(* CODESYS project OC_Core.library
   DefaultNamespace: OC_Core
   DocFormat: reStructuredText
   Description: Open Commissioning TwinCAT Core Library
   Author: SpiraTec AG
   Title: OC_Core
   Version: 1.1.0
   Company: Open Commissioning
   Placeholder: OC_Core

Project tree, tasks and I/O mapping:
  libraries: Tc2_Math, * (Beckhoff Automation GmbH); Tc2_Standard, * (Beckhoff Automation GmbH); Tc2_System, * (Beckhoff Automation GmbH); Tc2_Utilities, * (Beckhoff Automation GmbH); Tc3_Module, * (Beckhoff Automation GmbH); TcUnit, * (www.tcunit.org)
  Common/
    AdsMessageHandler/
      function block FB_AdsMessageHandler [ST]: bIsAdsMessageReadValid, bIsAdsMessageWriteValid, CreateAdsReadMessage, CreateAdsWriteMessage, LogAdsMessage, SendReadResponse, SendWriteResponse, stAdsMessageRead, stAdsMessageWrite
      data type ST_AdsMessage
    Components/
      function block FB_Clock [ST]
      function block FB_ClockAdvanced [ST]
      function block FB_DriveControl [ST]: bIsMoving, bIsPositionReached, fAccMax, fPosition, fPositionLimitMax, fPositionLimitMin, fTolerance, fVelocity, MoveAbsolute, MoveVelocity, Stop
      function block FB_Heater [ST]: FB_init, fValue, InitRun
      function block FB_MoveAbsolute [ST]: bIsReached, fPosition, fVelocity
      function block FB_MoveVelocity [ST]: bIsReached, fAcc, fVelocity
      function block FB_Ping [ST]: InitRun
    FileIo/
      data type E_FileIoState
      function block FB_FileIO [ST]: nBytesRead, nErrorId, Read, sNetId, sPath, Write
    Links/
      function block FB_LinkDataByte [ST]: GetLinkControlData, SetLinkStatusData
      function block FB_LinkDataDWord [ST]: GetLinkControlData, SetLinkStatusData
      function block FB_LinkDataLWord [ST]: GetLinkControlData, SetLinkStatusData
      function block FB_LinkDataReal [ST]: GetLinkControlData, SetLinkStatusData
      function block FB_LinkDataWord [ST]: GetLinkControlData, SetLinkStatusData
      function block FB_LinkDevice [ST]: GetControl, SetStatus
    RecordData/
      function block FB_RecordData [ST]: CmpIGrp, CmpInvokeId, CmpIOffs, DataValid, FB_init, GetReadIndication, GetWriteIndication, SendReadResponse, SendWriteResponse, Subscribe
      interface I_RecordData: GetReadIndication, GetWriteIndication, SendReadResponse, SendWriteResponse, Subscribe
      data type ST_RecordIdent
    System/
      data type E_ControllerType
      function F_IsSystemValid [ST]
      function F_LogError [ST]
      function F_LogMessage [ST]
      function F_LogWarning [ST]
      function block FB_Base [ST]
      function block FB_System [ST]: bDebug, bVerbose, eControllerType, fDeltaTime, fTimeScaling, InitRun
      global variables GVL_Core
    Utils/
      data type E_NetworkByteOrder
      function F_Clamp01 [ST]
      function F_Compare [ST]
      function F_GetHByte [ST]
      function F_GetLByte [ST]
      function F_InverBytesOrder [ST]
      function F_Norm [ST]
      function F_ScaleLREAL [ST]
      function F_Sign [ST]
      data type ST_ScaleConfig
  Devices/
    Basic/
      function block FB_Button [ST]
      function block FB_Cylinder [ST]
      function block FB_Device [ST]
      function block FB_DeviceByte [ST]
      function block FB_DeviceDWord [ST]
      function block FB_DeviceLWord [ST]
      function block FB_DeviceReal [ST]
      function block FB_DeviceWord [ST]
      function block FB_Drive [ST]
      function block FB_Lamp [ST]
      function block FB_Lock [ST]
      function block FB_Panel [ST]
      function block FB_Reader [ST]
      function block FB_Robot [ST]: ConnectJoints, GetJointsTarget, SetJointsStatus
      function block FB_SensorAnalog [ST]
      function block FB_SensorBinary [ST]
      function block FB_Switch [ST]
    Drives/
      Encoder/
        function block FB_Encoder [ST]: ControlLogic, InitRun
        data type ST_EncoderConfig
      FB_DS402/
        data type E_ControlMode
        data type E_DS402State
        function block FB_DS402 [ST]: AssignAddress, ControlLogic, eState, GetControlData, InitRun, PositionMode, SetStatusData, SpeedMode
        function block FB_DS402FSM [ST]: eState, IsDisableOperation, IsDisableVoltage, IsEnableOperation, IsFaultReset, IsQuickStop, IsShutdown, IsSwitchOn, nControl, nStatus, S0_NotReadyToSwitchOn, S1_SwitchOnDisabled, S2_ReadyToSwitchOn, S3_SwitchedOn, S4_OperationEnabled, S5_Fault, S6_FaultReactionActive, S7_QuickStopActive
        data type ST_DS402_6040h_ControlWord
        data type ST_DS402_6041h_StatusWord
        data type ST_DS402Config
      FB_SimMovidrive/
        data type E_SimMovidriveMode
        function block FB_SimMovidrivePDO12 [ST]: AssignProcessData, ControlLogic, GetControlData, GetControlMode, InitRun, SetStatusData
        data type ST_SimMovidriveConfig
        data type ST_SimMovidriveControlData
        data type ST_SimMovidriveStatusData
      FB_SimMovitrac/
        data type E_SimMovitracAssign
        function block FB_SimMovitrac [ST]: AssignProcessData, ControlLogic, GetControlData, InitRun, SetStatusData
        function block FB_SimMovitracB [ST]: AssignProcessData, ControlLogic, GetControlData, InitRun, SetStatusData
        function block FB_SimMovitracLTEB [ST]: ControlLogic, InitRun
        data type ST_SimMovitracConfig
        data type ST_SimMovitracControlData
        data type ST_SimMovitracStatusData
      FB_SimMovitracFSM/
        data type E_SimMovitracState
        function block FB_SimMovitracFSM [ST]: ControllerInhibit, Enable, Halt, HoldControl, nState, RapidStop
      FB_Starter/
        function block FB_Starter [ST]: AssignProcessData, ControlLogic, GetControlData, InitRun, SetStatusData
        data type ST_StarterConfig
        data type ST_StarterControlData
        data type ST_StarterStatusData
    Safety/
      function block FB_EuchnerMGB [ST]
      function block FB_EuchnerSTP [ST]
  Test/
    Common/
      function block FB_AdsMessageHandler_Test [ST]: TestCaseRead, TestCaseWrite
      function block FB_Clamp01_Test [ST]: TestCase
      function block FB_Compare_Test [ST]: TestCase
      function block FB_GetByte_Test [ST]: TestGetHByte, TestGetLByte
      function block FB_InverBytesOrder_Test [ST]: TestDWord, TestLWord, TestWord
      function block FB_Norm_Test [ST]: TestCase
      function block FB_RecordData_Test [ST]: TestAutoResponseReadMessage, TestAutoResponseWriteMessage, TestCaseCompare, TestCasesCompare, TestGetReadIndication, TestGetWriteIndication, TestSendReadResponse, TestSendWriteResponse
      function block FB_Scale_Test [ST]: TestCase, TestInputValidation
      function block FB_Sign_Test [ST]: TestCase
      function block FB_System_Test [ST]: TestInitialization, TestProperties
    Components/
      function block FB_DriveControl_Test [ST]: TestCaseMoveAbsolute, TestCaseMoveVelocity, TestCaseMoveVelocityLimits, TestProperties, TestStop
      function block FB_Heater_Test [ST]: TestLimits, TestState, TestValueChange
      function block FB_MoveAbsolute_Test [ST]: TestCaseMoveTo
      function block FB_MoveVelocity_Test [ST]: TestCaseMove
    Devices/
      function block FB_Button_Test [ST]
      function block FB_Cylinder_Test [ST]
      function block FB_Device_Test [ST]
      function block FB_DeviceByte_Test [ST]
      function block FB_DeviceDWord_Test [ST]
      function block FB_DeviceLWord_Test [ST]
      function block FB_DeviceReal_Test [ST]
      function block FB_DeviceWord_Test [ST]
      function block FB_Drive_Test [ST]
      function block FB_Lamp_Test [ST]
      function block FB_Lock_Test [ST]
      function block FB_Panel_Test [ST]
      function block FB_Reader_Test [ST]
      function block FB_Robot_Test [ST]: TestGetJoint, TestSetJoint
      function block FB_SensorAnalog_Test [ST]
      function block FB_SensorBinary_Test [ST]
      function block FB_Switch_Test [ST]
    Drives/
      function block FB_DS402_Test [ST]: EnableSequence, TestEnable, TestEnableSTO, TestPositionMode, TestSpeedDriveFactor, TestSpeedMode, TestSpeedModeEncoder, TestSpeedModeLinkOutput, TestSpeedModeModulo, TestSpeedModeOffset
      function block FB_DS402FSM_Test [ST]: GetDisableCommand, GetDisableVoltageCommand, GetEnableCommand, GetQuickStopCommand, GetShotdownCommand, GetSwitchOnCommand, TestEnableSequence, TestState_S0, TestState_S1, TestState_S2, TestState_S3, TestState_S4, TestState_S5, TestState_S6, TestState_S7
      function block FB_Encoder_Test [ST]: TestCase_Encoder
      function block FB_SimMovidriveFSM_Test [ST]: TestState
      function block FB_SimMovidrivePDO12_Test [ST]: Test_AssignProcessData, Test_GetControlData, Test_GetControlDataSWAP, Test_GetControlMode, Test_SetStatusData, Test_SetStatusDataSWAP
      function block FB_SimMovitrac_Test [ST]: Test_Movitrac
      function block FB_SimMovitracB_Test [ST]: TestCase_SimMovitracB
      function block FB_SimMovitracLTEB_Test [ST]: Test_DriveNotReady, Test_DriveReady, Test_DriveRunningBwd, Test_DriveRunningFwd
      function block FB_Starter_Test [ST]: Test_AssignProcessData, Test_DriveNoMovement, Test_DriveRunningCcw, Test_DriveRunningCw, Test_GetControlData, Test_GetControlDataSWAP, Test_SetStatusData, Test_SetStatusDataSWAP
    Safety/
      function block FB_Euchner_MGB_Test [ST]: Test_Button1, Test_Button2, Test_Button3, Test_Button4, Test_DoorClosed_Locked, Test_DoorClosed_NoLock, Test_DoorOpen, Test_Lamp1, Test_Lamp2, Test_Lamp3, Test_Lamp4
      function block FB_Euchner_STP_Test [ST]: Test_DoorClosedAndLocked, Test_DoorClosedAndUnlocked, Test_DoorOpen, Test_LampGN, Test_LampRD
    program PRG_TEST [ST]
*)

// Common/AdsMessageHandler/ST_AdsMessage
TYPE ST_AdsMessage :
STRUCT
	tNetID			: T_AmsNetID;
	tPort			: T_AmsPort;
	nInvokeID		: UDINT;
	nIdxGrp			: UDINT;
	nIdxOffs		: UDINT;
	nLength			: UDINT;
	nResult			: UDINT;
	aData			: ARRAY[0..239] OF BYTE;
END_STRUCT
END_TYPE

// Common/FileIo/E_FileIoState
{attribute 'conditionalshow'}
TYPE E_FileIoState :
(
	READY := 0,
	OPEN,
	CREATE,
	READ,
	WRITE,
	CLOSE,
	ERROR
);
END_TYPE

// Common/RecordData/ST_RecordIdent
TYPE ST_RecordIdent :
STRUCT
	nPort  			: T_AmsPort; //ADS-Port of the Profinet Device. Ignored when using PLCSIM Advanced
	nSlot			: UINT; //Slotnumber of the Profinet Device. Ignored when using PLCSIM Advanced
	nSubSlot		: UINT; //Subslotnumber of the Profinet Device. Ignored when using PLCSIM Advanced
	nPlcId			: UINT; //Identifier of the PLC when using PLCSIM Advanced
	nHardwareId		: UINT; //Hardware-ID of the device when using PLCSIM Advanced
END_STRUCT
END_TYPE

// Common/System/E_ControllerType
{attribute 'qualified_only'}
{attribute 'strict'}
TYPE E_ControllerType :
(
	NotDefined := 0,
	PlcSimAdvanced := 1
);
END_TYPE

// Common/Utils/E_NetworkByteOrder
{attribute 'qualified_only'}
{attribute 'strict'}
TYPE E_NetworkByteOrder :
(
	BigEndian := 0, //Big Endian (MOTOROLA)
	LittleEndian := 1 //Little Endian (Intel)	
);
END_TYPE

// Common/Utils/ST_ScaleConfig
{attribute 'pack_mode' := '0'} 
TYPE ST_ScaleConfig :
STRUCT
	fInputMin 	: LREAL := 0;
	fInputMax 	: LREAL := 100;
	fOutputMin 	: LREAL := 0;
	fOutputMax 	: LREAL := 65535;
END_STRUCT
END_TYPE

// Devices/Drives/Encoder/ST_EncoderConfig
TYPE ST_EncoderConfig :
STRUCT
	bIsIntegral   			: BOOL := FALSE;  //Integrate input value
	fNumerator 	  			: REAL := 0.0001; //[unit/INC]
	fDenominator  			: REAL := 1.0; 	// Scaling
	fModulo 	  			: REAL := 0; 	 	// Base divisor for modulo calculation [unit]; If not used set to 0.0	
	fInputFactor  			: REAL := 1.0; 
	fOutputFactor 			: REAL := 1.0;
	bInvertIncrementValue 	: BOOL;
END_STRUCT
END_TYPE

// Devices/Drives/FB_DS402/E_ControlMode
{attribute 'qualified_only'}
{attribute 'strict'}
TYPE E_ControlMode :
(
	Position 	:= 0,
	Speed	 	:= 1
)
BYTE;
END_TYPE

// Devices/Drives/FB_DS402/E_DS402State
{attribute 'qualified_only'}
{attribute 'strict'}
{attribute 'conditionalshow'}
TYPE E_DS402State :
(
	S0_NotReadyToSwitchOn,
	S1_SwitchOnDisabled,
	S2_ReadyToSwitchOn,
	S3_SwitchedOn,
	S4_OperationEnabled,
	S5_Fault,
	S6_FaultReactionActive,
	S7_QuickStopActive
);
END_TYPE

// Devices/Drives/FB_DS402/ST_DS402_6040h_ControlWord
{attribute 'pack_mode' := '1'}
TYPE ST_DS402_6040h_ControlWord :
STRUCT
	b0_SwitchOn 					: BIT;
	b1_EnableVoltage				: BIT;
	b2_QuickStop					: BIT;
	b3_EnableOperation				: BIT;
	b4_OperationModeSpecific		: BIT;
	b5_OperationModeSpecific		: BIT;
	b6_OperationModeSpecific		: BIT;
	b7_FaultReset					: BIT;
	b8_Reserved						: BIT;
	b9_Reserved						: BIT;
	b10_Reserved					: BIT;
	b11_Reserved					: BIT;
	b12_Reserved					: BIT;
	b13_Reserved					: BIT;
	b14_Reserved					: BIT;
	b15_Reserved					: BIT;
END_STRUCT
END_TYPE

// Devices/Drives/FB_DS402/ST_DS402_6041h_StatusWord
{attribute 'pack_mode' := '1'}
TYPE ST_DS402_6041h_StatusWord :
STRUCT
	b0_ReadyToSwitchOn 				: BIT; 
	b1_SwitchedOn 					: BIT; 
	b2_OperationEnabled 			: BIT; 
	b3_Fault						: BIT; 
	b4_VoltageEnabled				: BIT; 
	b5_QuickStop					: BIT;
	b6_SwitchOnDisabled				: BIT; 
	b7_Warning						: BIT; 
	b8_Synchranisation				: BIT; 
	b9_Remote						: BIT;
	b10_TargetReached				: BIT;
	b11_InternalLimitActive			: BIT; 
	b12_OperationModeSpecific		: BIT; 
	b13_OperationModeSpecific		: BIT; 
	b14_OperationModeSpecific		: BIT; 
	b15_ClosedLoopActive			: BIT;	
END_STRUCT
END_TYPE

// Devices/Drives/FB_DS402/ST_DS402Config
TYPE ST_DS402Config :
STRUCT	
	eControlMode 			: E_ControlMode := E_ControlMode.Position;
	eLinkControlMode 		: E_ControlMode := E_ControlMode.Position;
	fReferenceVelocity 		: REAL := 1000.0;
	fPositionOffset			: REAL := 0.0;	
	
	fEncoderNumerator		: REAL := 0.0001; //[unit/INC]
	fEncoderDenominator		: REAL := 1.0; //Scaling
	fEncoderModulo			: REAL := 0; //[unit]	
	
	fGearFactor				: REAL := 1.0;
	fEncoderOutputFactor	: REAL := 1.0;
	fLinkOutputFactor 		: REAL := 1.0;
	
	bSwapProcessData		: BOOL; //SWAP Process Data from/to FIELDBUS
END_STRUCT
END_TYPE

// Devices/Drives/FB_SimMovidrive/E_SimMovidriveMode
{attribute 'qualified_only'}
{attribute 'strict'}
TYPE E_SimMovidriveMode :
(
	Idle 	:= 0,
	Jog	 	:= 1,
	Ref		:= 2,
	Auto	:= 3
)BYTE;
END_TYPE

// Devices/Drives/FB_SimMovidrive/ST_SimMovidriveConfig
{attribute 'pack_mode' := '0'}
TYPE ST_SimMovidriveConfig :
STRUCT
	nSoftwareLimitMin	: DINT := -2147483648;	//Position limit minimum in LU
	nSoftwareLimitMax	: DINT := 2147483647;	//Position limit maximum in LU
	fDecCoastStop		: REAL := 10000.0;		//Deceleration for coast/brake stop in LU/s^2
	fDecRapidStop		: REAL := 10000.0;		//Deceleration for emergency stop in LU/s^2
	fDecRampStop		: REAL := 1000.0;		//Decceleration limit (bus stop) in LU/s^2
	fRatioVelocity		: REAL := 1.0;			//Ratio for setpoint velocity
	fRatioAccDec		: REAL := 1.0;			//Ratio for setpoint acceleration/deceleration
	fRatioPosition		: REAL := 0.001;		//Ratio for position output
	nJerk				: INT := 0;				//Jerk from 0 to 100%
	bSwapProcessData	: BOOL;					//SWAP Process Data from/to FIELDBUS
END_STRUCT
END_TYPE

// Devices/Drives/FB_SimMovidrive/ST_SimMovidriveControlData
{attribute 'pack_mode' := '1'}
TYPE ST_SimMovidriveControlData :
STRUCT
	bControllerInhibit		: BIT;	//0			0 = Enable, 1 = Inhibit controller, activate brake
	bRapidStop				: BIT;	//1			0 = Rapid stop, 1 = Enable
	bStop					: BIT;	//2			0 =  Stop at integrator ramp or process ramp, 1 = Enable
	bReserved3				: BIT;	//3			Currently not used
	bReserved4				: BIT;	//4			Currently not used
	bReserved5				: BIT;	//5			Currently not used
	bResetFAULT		  		: BIT;	//6			0 → 1 = Reset fault 
	bReserved7				: BIT;	//7			Currently not used	                            
	bStart					: BIT;	//8			1 = Enable Positioning / Referencing 
	bJog1					: BIT;	//9			1 = Enable Jog+
	bJog2					: BIT;	//10		1 = Enable Jog-
	bModeLow				: BIT;	//11		1 = Mode Jogging or Positioning (in combination with mode high)
	bModeHigh				: BIT;	//12		1 = Mode Referencing or Positioning (in combination with mode low)
	bReserved13				: BIT;	//13		Currently not used
	bReserved14				: BIT;	//14		Currently not used
	bReserved15				: BIT;	//15		Currently not used
	nTargetPosition			: DINT;	//16..47	Target position
	nVelocity				: UINT; //48..63	Velocity
	nAcceleration			: UINT; //64..79	Acceleration
	nDeceleration			: UINT; //80..95	Deceleration			
END_STRUCT
END_TYPE

// Devices/Drives/FB_SimMovidrive/ST_SimMovidriveStatusData
{attribute 'pack_mode' := '1'}
TYPE ST_SimMovidriveStatusData :
STRUCT
	bMotorTurning			: BIT;	//0			1 = Motor is turning
	bInverterReady			: BIT;	//1			1 = Inverter is ready
	bReferenced				: BIT;	//2			1 = Drive is referenced
	bTargetPositionReached	: BIT;	//3			1 = Target position reached
	bBrakeReleased			: BIT;	//4			1 = Brake is released
	bError					: BIT;	//5			1 = Error
	bLimitSwitchCW		  	: BIT;	//6			1 = Limit switch clock wise reached 
	bLimitSwitchCCW			: BIT;	//7			1 = Limit switch counter clock wise reached 	                            
	nStatus					: BYTE;	//8..15		Status / Errorcode
	nActPosition			: DINT; //16..47	Actual position
	nActVelocity			: UINT; //48..63	Actual velocity
	nActCurrent				: UINT; //64..79	Acutal current
	nActUnit				: UINT; //80..95	Actual unit utilization
END_STRUCT
END_TYPE

// Devices/Drives/FB_SimMovitrac/E_SimMovitracAssign
{attribute 'qualified_only'}
{attribute 'strict'}
TYPE E_SimMovitracAssign :
(
	ProcessData1 := 0,
	ProcessData2 := 2,
	ProcessData3 := 4,
	NoAssignment := 99
)DWORD;
END_TYPE

// Devices/Drives/FB_SimMovitrac/ST_SimMovitracConfig
TYPE ST_SimMovitracConfig :
STRUCT
	fDecCoastStop		: REAL := 200.0;	//Deceleration for coast/brake stop in ms. Reference speed is 3000 rpm.
	fDecRapidStop		: REAL := 500.0;	//Deceleration for emergency stop in ms. Reference speed is 3000 rpm.
	fProcessRamp		: REAL := 1000.0;	//Acc/Dec in ms when ramp via bus is not assigned. Reference speed is 3000 rpm.
	fGearFactor			: REAL := 1.0;		//Ratio for velocity output
	fReferenceVelocity	: REAL := 3000.0;

	nCtrlAssign			: E_SimMovitracAssign := E_SimMovitracAssign.ProcessData1; //Control word assignment
	nSpeedAssign		: E_SimMovitracAssign := E_SimMovitracAssign.ProcessData2; //Speed setpoint assignment
	nRampAssign			: E_SimMovitracAssign := E_SimMovitracAssign.NoAssignment; //Ramp setpoint assignment
	nStatusAssign		: E_SimMovitracAssign := E_SimMovitracAssign.ProcessData1; //Status word assignment
	nSpeedActAssign		: E_SimMovitracAssign := E_SimMovitracAssign.ProcessData2; //Actual speed assignment
	
	bSwapProcessData	: BOOL; //SWAP Process Data from/to FIELDBUS
END_STRUCT
END_TYPE

// Devices/Drives/FB_SimMovitrac/ST_SimMovitracControlData
{attribute 'pack_mode' := '1'}
TYPE ST_SimMovitracControlData :
STRUCT
	bControllerInhibit		: BIT;	//0			0 = Enable, 1 = Inhibit controller, activate brake
	bRapidStop				: BIT;	//1			0 = Rapid stop, 1 = Enable
	bStop					: BIT;	//2			0 =  Stop at integrator ramp or process ramp, 1 = Enable
	bReserved3				: BIT;	//3			Currently not used
	bReserved4				: BIT;	//4			Currently not used
	bReserved5				: BIT;	//5			Currently not used
	bResetFAULT		  		: BIT;	//6			0 → 1 = Reset fault 
	bReserved7				: BIT;	//7			Currently not used	                            
	bDirectionMotorPoti		: BIT;	//8			0 = CW, 1 = CCW 
	bMotorPotiUp			: BIT;	//9			1 = Increase poti value
	bMotorPotiDown			: BIT;	//10		1 = Decrease poti value
	bFixedInternalSetpoints	: BIT;	//11		1 = Fixed internal setpoints
	bFixedInternalSetp1		: BIT;	//12		1 = Fixed internal setpoint 1
	bFixedSetpSwitchover	: BIT;	//13		1 = Fixed setpoint switchover
	bReserved14				: BIT;	//14		Currently not used
	bReserved15				: BIT;	//15		Currently not used
	nSetpointSpeed			: INT; 	//			Setpoint speed in 0.2 rpm
	nRamp					: UINT; //			Ramp in ms			
END_STRUCT
END_TYPE

// Devices/Drives/FB_SimMovitrac/ST_SimMovitracStatusData
{attribute 'pack_mode' := '1'}
TYPE ST_SimMovitracStatusData :
STRUCT
	bEnableOutputStage		: BIT;	//0			1 = Output stage enabled
	bInverterReady			: BIT;	//1			1 = Inverter is ready
	bPoDataEnable			: BIT;	//2			1 = PO data enabled
	bReserved3				: BIT;	//3			Currently not used
	bReserved4				: BIT;	//4			Currently not used
	bError					: BIT;	//5			1 = Error
	bReserved6		  		: BIT;	//6			Currently not used
	bReserved7				: BIT;	//7			Currently not used
	nStatus					: BYTE;	//8..15		Status / Errorcode
	nActSpeed				: INT;	//			Actual speed in 0.2 rpm
END_STRUCT
END_TYPE

// Devices/Drives/FB_SimMovitracFSM/E_SimMovitracState
{attribute 'qualified_only'}
{attribute 'strict'}
{attribute 'conditionalshow'}
TYPE E_SimMovitracState :
(
	ControllerInhibit := 1,
	RapidStop := 2,
	Halt := 3,
	HoldControl := 4,
	Enable := 5
);
END_TYPE

// Devices/Drives/FB_Starter/ST_StarterConfig
{attribute 'pack_mode' := '1'}
TYPE ST_StarterConfig:
STRUCT
	fVelocity			: REAL := 100; 	// mm
	fAcceleration		: REAL := 500; 	// deg/s2
	fDeceleration		: REAL := 500; 	// deg/s2		
	bSwapProcessData	: BOOL; //SWAP Process Data from/to FIELDBUS
END_STRUCT
END_TYPE

// Devices/Drives/FB_Starter/ST_StarterControlData
{attribute 'pack_mode' := '1'}
TYPE ST_StarterControlData:
	STRUCT
		MotorCW           			: BIT; 		//0  
		MotorCCW	      			: BIT; 		//1  
		BrakeActuation				: BIT; 		//2  
		TripReset          			: BIT; 		//3  
		EmergStart        			: BIT; 		//4  
		SelfTest	      			: BIT; 		//5  
		Reserve06          			: BIT; 		//6  
		Reserve07		   			: BIT; 		//7 
		Reserve10		   			: BIT; 		//08  
		Reserve11		   			: BIT; 		//09  
		Reserve12		   			: BIT; 		//10  
		Reserve13		   			: BIT; 		//11  
		Reserve14		   			: BIT; 		//12  
		Reserve15		   			: BIT; 		//13  
		Reserve16		   			: BIT; 		//14  
		DisQuickStop	   			: BIT; 		//15   
	END_STRUCT
END_TYPE

// Devices/Drives/FB_Starter/ST_StarterStatusData
{attribute 'pack_mode' := '1'}
TYPE ST_StarterStatusData:
	STRUCT
		Ready           			: BIT; 		//0  
		MotorON		      			: BIT; 		//1  
		GroupFault					: BIT; 		//2  
		GroupWarn          			: BIT; 		//3  
		Input1	        			: BIT; 		//4  
		Input2		      			: BIT; 		//5  
		Input3          			: BIT; 		//6  
		Input4			   			: BIT; 		//7 
		MotorCurrent0	   			: BIT; 		//08  
		MotorCurrent1	   			: BIT; 		//09  
		MotorCurrent2	   			: BIT; 		//10  
		MotorCurrent3	   			: BIT; 		//11  
		MotorCurrent4	   			: BIT; 		//12  
		MotorCurrent5	   			: BIT; 		//13  
		ManualLocalMode	   			: BIT; 		//14  
		RampOperation	   			: BIT; 		//15  
	END_STRUCT
END_TYPE

// Common/System/GVL_Core
{attribute 'qualified_only'}
{attribute 'conditionalshow'}
VAR_GLOBAL	
	refSystem 			: REFERENCE TO FB_System;		
END_VAR

// Common/AdsMessageHandler/FB_AdsMessageHandler
(*ADS Message Handler is responsible for indication of the ADS Read/Write messages for local NetId and generation of the response message*)
FUNCTION_BLOCK FB_AdsMessageHandler
VAR_INPUT
	bDisable 				: BOOL;	//Deactivate cyclical execution
	bLog					: BOOL;	//Log ADS messages data in the console
	bVerbose				: BOOL; //Log Verbose information in the console
END_VAR

VAR	
	fbAdsWriteIndicator 	: AdsWriteInd;	
	fbAdsReadIndicator 		: AdsReadInd;
	fbAdsWriteResponse		: AdsWriteRes;
	fbAdsReadResponse		: AdsReadRes;	
	_stAdsMessageWrite		: ST_AdsMessage;
	_stAdsMessageRead		: ST_AdsMessage;	
	
    sFormatReciveWrite		: STRING := 'AdsWriteInd Port: %X, IdxGrp: %X, IdxOffs: %X, InvokeId %X, Length: %X';
	sFormatReciveRead		: STRING := 'AdsReadInd Port: %X, IdxGrp: %X, IdxOffs: %X, InvokeId %X, Length: %X';
	sFormatResponseWrite	: STRING := 'AdsWriteRes Port: %X, IdxGrp: %X, IdxOffs: %X, InvokeId %X, Length: %X';
	sFormatResponseRead		: STRING := 'AdsReadRes Port: %X, IdxGrp: %X, IdxOffs: %X, InvokeId %X, Length: %X';  
END_VAR

IF bDisable THEN RETURN; END_IF

//Reset Indication and Result FBs
fbAdsWriteResponse(RESPOND := FALSE);
fbAdsReadResponse(RESPOND := FALSE);

//Capture all Write requests
fbAdsWriteIndicator();
CreateAdsWriteMessage();
		
//Capture all Read requests
fbAdsReadIndicator();
CreateAdsReadMessage();

(*Returns the status of the indication of the read message in the current frame*)
PROPERTY PUBLIC bIsAdsMessageReadValid : BOOL
GET
bIsAdsMessageReadValid := _stAdsMessageRead.tPort <> 0;
END_GET
END_PROPERTY

(*Returns the status of the indication of the write message in the current frame*)
PROPERTY PUBLIC bIsAdsMessageWriteValid : BOOL
GET
bIsAdsMessageWriteValid := _stAdsMessageWrite.tPort <> 0;
END_GET
END_PROPERTY

METHOD PRIVATE CreateAdsReadMessage : BOOL
IF NOT fbAdsReadIndicator.VALID THEN RETURN; END_IF

MEMSET(ADR(_stAdsMessageRead), 0, SIZEOF(ST_AdsMessage));
_stAdsMessageRead.tNetId 		:= fbAdsReadIndicator.NETID;
_stAdsMessageRead.tPort 		:= fbAdsReadIndicator.PORT;
_stAdsMessageRead.nInvokeId 	:= fbAdsReadIndicator.INVOKEID;
_stAdsMessageRead.nIdxGrp 		:= fbAdsReadIndicator.IDXGRP;
_stAdsMessageRead.nIdxOffs 		:= fbAdsReadIndicator.IDXOFFS;
_stAdsMessageRead.nLength 		:= fbAdsReadIndicator.LENGTH;

IF bVerbose THEN
	LogAdsMessage(_stAdsMessageWrite, sFormatReciveRead);
END_IF

fbAdsReadIndicator(CLEAR := TRUE);
fbAdsReadIndicator(CLEAR := FALSE);
END_METHOD

METHOD PRIVATE CreateAdsWriteMessage : BOOL
IF NOT fbAdsWriteIndicator.VALID THEN RETURN; END_IF

MEMSET(ADR(_stAdsMessageWrite), 0, SIZEOF(ST_AdsMessage));
_stAdsMessageWrite.tNetId 		:= fbAdsWriteIndicator.NETID;
_stAdsMessageWrite.tPort 		:= fbAdsWriteIndicator.PORT;
_stAdsMessageWrite.nInvokeId 	:= fbAdsWriteIndicator.INVOKEID;
_stAdsMessageWrite.nIdxGrp 		:= fbAdsWriteIndicator.IDXGRP;
_stAdsMessageWrite.nIdxOffs 	:= fbAdsWriteIndicator.IDXOFFS;
_stAdsMessageWrite.nLength 		:= fbAdsWriteIndicator.LENGTH;
			
//Limit size to 240
IF _stAdsMessageWrite.nLength > 240 THEN
	IF bVerbose THEN
		F_LOGWARNING(CONCAT('WRREC data length limited to 240. Requested data length was ', TO_STRING(_stAdsMessageWrite.nLength)));
	END_IF
	_stAdsMessageWrite.nLength := 240;
END_IF

MEMCPY(ADR(_stAdsMessageWrite.aData), fbAdsWriteIndicator.DATAADDR, _stAdsMessageWrite.nLength);

IF bVerbose THEN
	LogAdsMessage(_stAdsMessageWrite, sFormatReciveWrite);
END_IF

fbAdsWriteIndicator(CLEAR := TRUE);
fbAdsWriteIndicator(CLEAR := FALSE);
END_METHOD

METHOD PRIVATE LogAdsMessage : BOOL
VAR_INPUT
	stAdsMessage 			: ST_AdsMessage;
	sFormat 				: STRING;
END_VAR

VAR
	fbFormatString			: FB_FormatString2;
	sMessage				: STRING;
END_VAR
fbFormatString(
	pFormatString := ADR(sFormat),
	arg1 := F_UINT(stAdsMessage.tPort),
	arg2 := F_UDINT(stAdsMessage.nIdxGrp),
	arg3 := F_UDINT(stAdsMessage.nIdxOffs),		
	arg4 := F_UDINT(stAdsMessage.nInvokeID),
	arg5 := F_UDINT(stAdsMessage.nLength),
	pDstString := ADR(sMessage),
	nDstSize := SIZEOF(sMessage));
F_LogMessage(sMessage);
END_METHOD

(*Send ADS Read Response message*)
METHOD PUBLIC SendReadResponse : HRESULT
VAR_INPUT
	stAdsMessage 	: ST_AdsMessage; //Response ADS Message
END_VAR
IF fbAdsReadResponse.RESPOND THEN
	SendReadResponse := S_PENDING;
	RETURN;
END_IF

//Limit size to 240
IF stAdsMessage.nLength > 240 THEN
	IF bVerbose THEN
		F_LOGWARNING(CONCAT('RDRES data length limited to 240. Requested data length was ', TO_STRING(stAdsMessage.nLength)));
	END_IF
	stAdsMessage.nLength := 240;
END_IF

fbAdsReadResponse(
	NETID:= stAdsMessage.tNetId, 
	PORT:= stAdsMessage.tPort, 
	INVOKEID:= stAdsMessage.nInvokeId, 
	RESULT:= stAdsMessage.nResult, 
	LEN:= stAdsMessage.nLength,
	DATAADDR:= ADR(stAdsMessage.aData),
	RESPOND:= TRUE);
IF bVerbose OR bLog THEN	
	LogAdsMessage(stAdsMessage, sFormatResponseRead);
END_IF

SendReadResponse := S_OK;
END_METHOD

(*Send ADS Read Response message*)
METHOD PUBLIC SendWriteResponse : HRESULT
VAR_INPUT
	stAdsMessage 	: ST_AdsMessage; //Response ADS Message
END_VAR
IF fbAdsWriteResponse.RESPOND THEN
	SendWriteResponse := S_PENDING;
	RETURN;
END_IF

fbAdsWriteResponse(
	NETID:= stAdsMessage.tNetId, 
	PORT:= stAdsMessage.tPort, 
	INVOKEID:= stAdsMessage.nInvokeId, 
	RESULT:= stAdsMessage.nResult, 
	RESPOND:= TRUE);	

IF bVerbose OR bLog THEN		
	LogAdsMessage(stAdsMessage, sFormatResponseWrite);
END_IF
	
SendWriteResponse := S_OK;
END_METHOD

(*Get last valid ADS Read Message*)
PROPERTY stAdsMessageRead : REFERENCE TO ST_AdsMessage
GET
stAdsMessageRead REF= _stAdsMessageRead;
END_GET
END_PROPERTY

(*Get last valid ADS Write Message*)
PROPERTY stAdsMessageWrite : REFERENCE TO ST_AdsMessage
GET
stAdsMessageWrite REF= _stAdsMessageWrite;
END_GET
END_PROPERTY

END_FUNCTION_BLOCK

// Common/System/F_LogWarning
{attribute 'hide_all_locals'}
FUNCTION F_LogWarning : BOOL
VAR_INPUT
	sMessage : T_MAXSTRING;
END_VAR

VAR CONSTANT	
	LOGHEADER		: T_MAXSTRING := 'Open Commissioning: %s';
END_VAR

ADSLOGSTR(ADSLOG_MSGTYPE_WARN, LOGHEADER, sMessage);

END_FUNCTION

// Common/System/F_LogMessage
{attribute 'hide_all_locals'}
FUNCTION F_LogMessage : BOOL
VAR_INPUT
	sMessage : T_MAXSTRING;
END_VAR

VAR CONSTANT	
	LOGHEADER		: T_MAXSTRING := 'Open Commissioning: %s';
END_VAR

ADSLOGSTR(ADSLOG_MSGTYPE_HINT, LOGHEADER, sMessage);

END_FUNCTION

// Common/Components/FB_Clock
FUNCTION_BLOCK FB_Clock
VAR_INPUT
	tPT		: TIME;
END_VAR

VAR_OUTPUT
	bQ		: BOOL;
END_VAR

VAR
	fbTon1	: TON;
	fbTon2	: TON;
END_VAR

fbTon1.PT := tPT;
fbTon2.PT := tPT;

fbTon1(IN := NOT bQ);
fbTon2(IN := bQ);

IF fbTon1.Q THEN
	bQ := TRUE;
END_IF

IF fbTon2.Q THEN
	bQ := FALSE;
END_IF

END_FUNCTION_BLOCK

// Common/Components/FB_ClockAdvanced
FUNCTION_BLOCK FB_ClockAdvanced
VAR_INPUT
	bEnable				: BOOL;
	tHighImpulsePT		: TIME;
	tLowImpulsePT		: TIME;
	tDelay				: TIME;
	bInvert				: BOOL;
END_VAR

VAR_OUTPUT
	bQ					: BOOL;
END_VAR

VAR
	fbTon1				: TON;
	fbTon2				: TON;
	fbTonDelay 			: TON;
	bLocalGenerator 	: BOOL;
END_VAR

fbTonDelay.IN := bEnable;
fbTonDelay.PT := tDelay;
fbTonDelay();

IF NOT bEnable THEN
	bQ := FALSE;
	fbTon1(IN := FALSE);
	fbTon2(IN := FALSE);
	RETURN;
END_IF

IF fbTonDelay.Q THEN
	IF bInvert THEN
		fbTon1.PT := tHighImpulsePT;
		fbTon2.PT := tLowImpulsePT;
	ELSE
		fbTon1.PT := tLowImpulsePT;
		fbTon2.PT := tHighImpulsePT;
	END_IF
	
	fbTon1(IN := NOT bLocalGenerator);
	fbTon2(IN := bLocalGenerator);
	
	IF fbTon1.Q THEN
		bLocalGenerator := TRUE;
	END_IF
	
	IF fbTon2.Q THEN
		bLocalGenerator := FALSE;
	END_IF
	
	bQ := bLocalGenerator;
	
	IF bInvert THEN
		bQ := NOT bLocalGenerator;
	END_IF
	
END_IF

END_FUNCTION_BLOCK

// Common/Components/FB_DriveControl
{attribute 'conditionalshow_all_locals'}
FUNCTION_BLOCK INTERNAL FB_DriveControl
VAR
	_fPosition 				: REAL;
	_fVelocity 				: REAL;		
	_bIsPositionReached 	: BOOL := TRUE;		
	
	_fPositionLimitMin 		: REAL := -1E+12;
	_fPositionLimitMax 		: REAL := 1E+12;
	_fAccMax				: REAL := 1E+12;	
	_fTolerance				: REAL := 1E-6;
	
	fbMoveAbsolute 			: FB_MoveAbsolute();
	fbMoveVelocity			: FB_MoveVelocity();
END_VAR

PROPERTY bIsMoving : BOOL
GET
bIsMoving := NOT F_Compare(_fVelocity, 0, 1E-3);
END_GET
END_PROPERTY

PROPERTY bIsPositionReached : BOOL
GET
bIsPositionReached := _bIsPositionReached;
END_GET
END_PROPERTY

PROPERTY fAccMax : REAL
GET
fAccMax := _fAccMax;
END_GET
SET
_fAccMax := fAccMax;
END_SET
END_PROPERTY

PROPERTY fPosition : REAL
GET
fPosition := _fPosition;
END_GET
SET
_fPosition := fPosition;
END_SET
END_PROPERTY

PROPERTY fPositionLimitMax : REAL
GET
fPositionLimitMax := _fPositionLimitMax;
END_GET
SET
_fPositionLimitMax := fPositionLimitMax;
END_SET
END_PROPERTY

PROPERTY fPositionLimitMin : REAL
GET
fPositionLimitMin := _fPositionLimitMin;
END_GET
SET
_fPositionLimitMin := fPositionLimitMin;
END_SET
END_PROPERTY

PROPERTY fTolerance : REAL
GET
fTolerance := _fTolerance;
END_GET
SET
_fTolerance := fTolerance;
END_SET
END_PROPERTY

PROPERTY fVelocity : REAL
GET
fVelocity := _fVelocity;
END_GET
SET
_fVelocity := fVelocity;
END_SET
END_PROPERTY

METHOD INTERNAL MoveAbsolute
VAR_INPUT
	fPosition 			: REAL;
	fVelocity			: REAL;
	fAcceleration		: REAL;
	fDeceleration   	: REAL;
END_VAR
fbMoveAbsolute.fPosition := _fPosition;
fbMoveAbsolute.fVelocity := _fVelocity;

fbMoveAbsolute(
	fTargetPosition := LIMIT(_fPositionLimitMin, fPosition, _fPositionLimitMax),
	fTargetVelocity := fVelocity,
	fAccMax := fAcceleration,
	fDecMax := fDeceleration,
	fTolerance := _fTolerance);					

_fVelocity := fbMoveAbsolute.fVelocity;
_fPosition := fbMoveAbsolute.fPosition;

_bIsPositionReached := F_Compare(fPosition, _fPosition, _fTolerance);
END_METHOD

METHOD INTERNAL MoveVelocity
VAR_INPUT
	fVelocity 			: REAL;
	fAcceleration 		: REAL;
	fDeceleration 		: REAL;
END_VAR
fbMoveVelocity.fVelocity := _fVelocity;
fbMoveVelocity.fTargetVelocity := fVelocity;
fbMoveVelocity.fAccMax := fAcceleration;
fbMoveVelocity.fDecMax := fDeceleration;	
	
IF _fPositionLimitMax <> 0 AND _fPositionLimitMin <> 0 THEN
	IF _fPosition >= _fPositionLimitMax OR _fPosition <= _fPositionLimitMin THEN
		fbMoveVelocity.fTargetVelocity := 0;
		fbMoveVelocity.fAccMax := _fAccMax;
		fbMoveVelocity.fDecMax := _fAccMax;
	END_IF		
END_IF
	
fbMoveVelocity();
	
_fVelocity := fbMoveVelocity.fVelocity;	

_fPosition := _fPosition + _fVelocity * GVL_Core.fbSystem.fDeltaTime * GVL_Core.fbSystem.fTimeScaling;
_bIsPositionReached := F_Compare(fPosition, _fPosition, _fTolerance);
END_METHOD

METHOD INTERNAL Stop
VAR_INPUT
	fDeceleration 	: REAL; 
END_VAR

VAR
	fSign 			: REAL;
	fTolerance 		: REAL := 1E-3;
	fAbsVelocity 	: REAL;
END_VAR
fSign := F_Sign(_fVelocity);
fAbsVelocity := ABS(_fVelocity);

IF fAbsVelocity > fTolerance THEN
	fAbsVelocity := fAbsVelocity - ABS(fDeceleration) * GVL_Core.fbSystem.fDeltaTime * GVL_Core.fbSystem.fTimeScaling;
	fAbsVelocity := LIMIT(0, fAbsVelocity, 3.402823E+38);
	_fVelocity := fAbsVelocity * fSign;	
ELSE
	_fVelocity := 0;
END_IF
END_METHOD

END_FUNCTION_BLOCK

// Common/Components/FB_MoveAbsolute
FUNCTION_BLOCK INTERNAL FB_MoveAbsolute 
VAR_INPUT
	fTargetPosition 	: REAL;
	fTargetVelocity 	: REAL; 
	fAccMax 			: REAL; 
	fDecMax 			: REAL;	
	fTolerance			: REAL := 1E-6;	
END_VAR

VAR
	_fVelocity 			: REAL;
	_fPosition 			: REAL;
	_bIsReached			: BOOL;
END_VAR

fTargetVelocity := ABS(fTargetVelocity); 
fAccMax := ABS(fAccMax);
fDecMax := -ABS(fDecMax);

IF F_Compare(fTargetPosition, _fPosition, fTolerance) THEN
	_fVelocity := 0;
	_fPosition := fTargetPosition;
	_bIsReached := TRUE;	
ELSE
	(* Calculate velocity and position *)
	IF fTargetPosition > _fPosition THEN		
		IF _fVelocity < 0 THEN
			_fVelocity := MIN(_fVelocity - fDecMax * GVL_Core.fbSystem.fDeltaTime * GVL_Core.fbSystem.fTimeScaling, fTargetVelocity);
		ELSE
			IF _fVelocity > fTargetVelocity THEN
				_fVelocity := MAX(_fVelocity + fDecMax * GVL_Core.fbSystem.fDeltaTime * GVL_Core.fbSystem.fTimeScaling, fTargetVelocity);
			ELSE
				_fVelocity := MIN(_fVelocity + fAccMax * GVL_Core.fbSystem.fDeltaTime * GVL_Core.fbSystem.fTimeScaling, fTargetVelocity);
			END_IF

			_fVelocity := MIN(SQRT((_fPosition - fTargetPosition) * 2.0 * fDecMax - 1.5 * GVL_Core.fbSystem.fDeltaTime * GVL_Core.fbSystem.fTimeScaling * fDecMax), _fVelocity);
		END_IF

		_fPosition := _fPosition + MIN(_fVelocity * GVL_Core.fbSystem.fDeltaTime * GVL_Core.fbSystem.fTimeScaling, fTargetPosition - _fPosition);	
	ELSE		
		IF _fVelocity > 0 THEN
			_fVelocity := MAX(_fVelocity + fDecMax * GVL_Core.fbSystem.fDeltaTime * GVL_Core.fbSystem.fTimeScaling, -fTargetVelocity);
		ELSE
			IF _fVelocity < -fTargetVelocity THEN
				_fVelocity := MIN(_fVelocity - fDecMax * GVL_Core.fbSystem.fDeltaTime * GVL_Core.fbSystem.fTimeScaling, -fTargetVelocity);
			ELSE				
				_fVelocity := MAX(_fVelocity - fAccMax * GVL_Core.fbSystem.fDeltaTime * GVL_Core.fbSystem.fTimeScaling, -fTargetVelocity);
			END_IF
			
			_fVelocity := MAX(-SQRT((_fPosition - fTargetPosition) * 2.0 * -fDecMax - 1.5 * GVL_Core.fbSystem.fDeltaTime * GVL_Core.fbSystem.fTimeScaling * fDecMax), _fVelocity);
	   END_IF

		_fPosition := _fPosition + MAX(_fVelocity * GVL_Core.fbSystem.fDeltaTime * GVL_Core.fbSystem.fTimeScaling, fTargetPosition - _fPosition);	
	END_IF;
	
	_bIsReached := FALSE;		
END_IF;

PROPERTY bIsReached : BOOL
GET
bIsReached := THIS^._bIsReached;
END_GET
END_PROPERTY

PROPERTY fPosition : REAL
GET
fPosition := _fPosition;
END_GET
SET
_fPosition := fPosition;
END_SET
END_PROPERTY

PROPERTY fVelocity : REAL
GET
fVelocity := _fVelocity;
END_GET
SET
_fVelocity := fVelocity;
END_SET
END_PROPERTY

END_FUNCTION_BLOCK

// Common/Utils/F_Compare
{attribute 'hide_all_locals'}
FUNCTION F_Compare : BOOL
VAR_INPUT
	fValueA 		: REAL;
	fValueB 		: REAL;
	fTolerance 		: REAL := 1E-6;	
END_VAR

VAR
	fDifference 	: REAL;
END_VAR

fDifference := ABS(fValueB - fValueA);
fTolerance := LIMIT(1E-6, ABS(fTolerance), 1E+6);
F_Compare := fTolerance > fDifference;

END_FUNCTION

// Common/Components/FB_MoveVelocity
FUNCTION_BLOCK INTERNAL FB_MoveVelocity
VAR_INPUT
	fTargetVelocity 	: REAL;
	fAccMax 			: REAL;
	fDecMax 			: REAL;
END_VAR

VAR
	_fVelocity 			: REAL;	
	_fAcc 				: REAL;
	_bIsReached			: BOOL;
	fVelocityTolerance	: REAL;
END_VAR

_bIsReached := FALSE;
IF _fAcc = 0 THEN
	IF ABS(fAccMax) > ABS(fDecMax) THEN
		fVelocityTolerance := ABS(fAccMax) * GVL_Core.fbSystem.fDeltaTime * GVL_Core.fbSystem.fTimeScaling;
	ELSE
		fVelocityTolerance := ABS(fDecMax) * GVL_Core.fbSystem.fDeltaTime * GVL_Core.fbSystem.fTimeScaling;
	END_IF
ELSE
	fVelocityTolerance := ABS(_fAcc) * GVL_Core.fbSystem.fDeltaTime * GVL_Core.fbSystem.fTimeScaling;
END_IF	

(* Calculate acceleration *)
//Hold velocity (velocity reached)
IF F_Compare(fVelocity, fTargetVelocity, fVelocityTolerance) THEN
	_fAcc := 0;
	_fVelocity := fTargetVelocity;
	_bIsReached := TRUE;
	RETURN;
END_IF

IF _fVelocity - fTargetVelocity > fVelocityTolerance THEN
	//Decelerate
	IF _fVelocity < 0 THEN
		_fAcc := -ABS(fAccMax);
	ELSE
		_fAcc := -ABS(fDecMax);
	END_IF
 ELSIF _fVelocity - fTargetVelocity < -fVelocityTolerance THEN
	//Accelerate
	IF _fVelocity < 0 THEN
		_fAcc := ABS(fDecMax);
	ELSE
		_fAcc := ABS(fAccMax);
	END_IF
END_IF

_fVelocity := _fVelocity + _fAcc * GVL_Core.fbSystem.fDeltaTime * GVL_Core.fbSystem.fTimeScaling;
_bIsReached := F_Compare(_fVelocity, fTargetVelocity, fVelocityTolerance);

PROPERTY bIsReached : BOOL
GET
bIsReached := THIS^._bIsReached;
END_GET
END_PROPERTY

PROPERTY fAcc : REAL
GET
fAcc := THIS^._fAcc;
END_GET
SET
THIS^._fAcc := fAcc;
END_SET
END_PROPERTY

PROPERTY fVelocity : REAL
GET
fVelocity := THIS^._fVelocity;
END_GET
SET
THIS^._fVelocity := fVelocity;
END_SET
END_PROPERTY

END_FUNCTION_BLOCK

// Common/Utils/F_Sign
{attribute 'hide_all_locals'}
FUNCTION F_Sign : REAL
VAR_INPUT
	fValue 	: REAL;
END_VAR

IF (fValue >= 0) THEN
	F_Sign := 1;
ELSE
	F_Sign := -1;	
END_IF

END_FUNCTION

// Common/Components/FB_Heater
FUNCTION_BLOCK FB_Heater
VAR_INPUT
	bEnable 		: BOOL;	
	fHeatingSpeed 	: REAL := 1; //[*/s]
	fCoolingSpeed 	: REAL := 1; //[*/s]
	fLimitMin 		: REAL := 0; //[*]
	fLimitMax 		: REAL := 100; //[*]
	fInitValue 		: REAL; //[*]
END_VAR

VAR_OUTPUT
	bEnabled 		: BOOL;
	bIsLimitMin		: BOOL;
	bIsLimitMax		: BOOL;	
END_VAR

VAR
	_fValue 		: REAL; //[*]
END_VAR

InitRun();

bEnabled := bEnable;

_fValue := _fValue - fCoolingSpeed * GVL_Core.fbSystem.fDeltaTime;

IF bEnable THEN
	_fValue := _fValue + fHeatingSpeed * GVL_Core.fbSystem.fDeltaTime;
END_IF

bIsLimitMin := _fValue <= fLimitMin;
bIsLimitMax := _fValue >= fLimitMax;
_fValue := LIMIT(fLimitMin, _fValue, fLimitMax);

METHOD FB_init : BOOL
VAR_INPUT
	bInitRetains : BOOL := TRUE; // if TRUE, the retain variables are initialized (warm start / cold start)
	bInCopyCode : BOOL;  // if TRUE, the instance afterwards gets moved into the copy code (online change)
	fInitValue : REAL;
END_VAR
fValue := fInitValue;
END_METHOD

PROPERTY fValue : REAL
GET
fValue := _fValue;
END_GET
SET
_fValue := fValue;
END_SET
END_PROPERTY

METHOD INTERNAL InitRun
VAR_INST
	bInitRun : BOOL := TRUE;
END_VAR
IF NOT bInitRun THEN RETURN; END_IF
bInitRun := FALSE;
END_METHOD

END_FUNCTION_BLOCK

// Common/Components/FB_Ping
FUNCTION_BLOCK FB_Ping
VAR_INPUT	
	bFeedback 		: BOOL;	// bit from unity status
END_VAR

VAR_OUTPUT
	bTrigger		: BOOL;	// bit to unity control
	nActET			: DWORD;  // elapsed time in ms
	nMaxET			: DWORD;  // max. elapsed time in ms
END_VAR

VAR	
	bEnable			: BOOL;
	fbTrigStart		: R_TRIG;
	fbTrigStop		: R_TRIG;
	fbTrigRestart 	: F_TRIG;
	nTimeStart 		: TIME;
	nTimeStop 		: TIME;
END_VAR

InitRun();

fbTrigStart(CLK := bEnable);
fbTrigStop(CLK := bFeedback);
fbTrigRestart(CLK := bFeedback);

IF fbTrigStart.Q OR fbTrigRestart.Q THEN
	nActET := 0;
	bTrigger := TRUE;
	nTimeStart := TIME();
END_IF


IF fbTrigStop.Q THEN
	bTrigger := FALSE;
	nTimeStop := TIME();
	nActET := TIME_TO_DWORD(nTimeStop - nTimeStart);
	IF nActET >= nMaxET THEN
		nMaxET := nActET;
	END_IF
END_IF

METHOD INTERNAL InitRun
VAR_INST
	bInitRun : BOOL := TRUE;
END_VAR
IF NOT bInitRun THEN RETURN; END_IF

bInitRun := FALSE;
nActET := 0;
nMaxET := 0;
END_METHOD

END_FUNCTION_BLOCK

// Common/FileIo/FB_FileIO
FUNCTION_BLOCK FB_FileIO
VAR	
	_sNetId				: STRING;
	_sPath				: STRING;
	fbFileOpen 			: FB_FileOpen;
	fbFileWrite 		: FB_FileWrite;
	fbFileRead 			: FB_FileRead;
	fbFileClose 		: FB_FileClose;	
	fbCreateDir			: FB_CreateDir;
	nHFile 				: UINT := 0;
	eReadState 			: E_FileIoState := READY;
	eWriteState 		: E_FileIoState := READY;
	nBytesReadResult	: UDINT;
	nErrorIdResult		: UDINT;	
END_VAR

PROPERTY PUBLIC nBytesRead : UDINT
GET
nBytesRead := nBytesReadResult;
END_GET
SET
PRIVATE
nBytesReadResult := nBytesRead;
END_SET
END_PROPERTY

PROPERTY PUBLIC nErrorId : uDINT
GET
nErrorId := nErrorIdResult;
END_GET
SET
PRIVATE
nErrorIdResult := nErrorId;
END_SET
END_PROPERTY

METHOD PUBLIC Read : BOOL
VAR_INPUT
	sFileName	: T_MaxString;
	pData		: PVOID;
	nLength		: UDINT;
END_VAR
Read := FALSE;
CASE eReadState OF
	E_FileIoState.READY:
		fbFileOpen(sNetId := _sNetId, bExecute := FALSE);
		fbFileRead(sNetId := _sNetId, bExecute := FALSE);
		fbFileClose(sNetId := _sNetId, bExecute := FALSE);
		eReadState := E_FileIoState.OPEN;
		
	E_FileIoState.OPEN:
		nErrorId := 0;
		nBytesRead := 0;
		IF nHFile = 0 THEN
			fbFileOpen.sPathName := sFileName;
			fbFileOpen.nMode := FOPEN_MODEREAD;
			fbFileOpen.ePath := PATH_GENERIC;
			fbFileOpen(bExecute := TRUE);
		END_IF
		IF fbFileOpen.hFile <> 0 AND NOT fbFileOpen.bBusy AND NOT fbFileOpen.bError THEN
			nHFile := fbFileOpen.hFile;
			fbFileOpen(bExecute := FALSE);			
			fbFileRead.hFile := nHFile;
			fbFileRead.cbReadLen := nLength;
			fbFileRead.pReadBuff := pData;
			eReadState := E_FileIoState.READ;
		END_IF
		IF fbFileOpen.bError THEN
			fbFileOpen(bExecute := FALSE);
			nErrorId := fbFileOpen.nErrId;
			eReadState := E_FileIoState.CREATE;
		END_IF
		
	E_FileIoState.CREATE:
		IF THIS^.Write(sFileName, pData, nLength) THEN
			IF nErrorId = 0 THEN
				eReadState := E_FileIoState.OPEN;
			ELSE
				eReadState := E_FileIoState.ERROR;
			END_IF
		END_IF
				
	E_FileIoState.READ:
		fbFileRead(bExecute := TRUE);
		IF NOT fbFileRead.bBusy AND NOT fbFileRead.bError THEN
			nBytesRead := fbFileRead.cbRead;
			fbFileRead(bExecute := FALSE);
			eReadState := E_FileIoState.CLOSE;
		END_IF
		IF fbFileRead.bError THEN
			nErrorId := fbFileRead.nErrId;
			eReadState := E_FileIoState.ERROR;
		END_IF
		
	E_FileIoState.CLOSE:
		IF nHFile <> 0 THEN
			fbFileClose(hFile := nHFile, bExecute := TRUE);
		END_IF
		IF NOT fbFileClose.bBusy THEN
			fbFileClose(bExecute := FALSE);
			nHFile := 0;
			eReadState := E_FileIoState.READY;
			Read := TRUE;
		END_IF
				
	E_FileIoState.ERROR:
		F_LogError(CONCAT('Error reading/writing file in ', CONCAT(_sNetId, CONCAT(' - ', _sPath))));
		eReadState := E_FileIoState.CLOSE;
		
END_CASE
END_METHOD

PROPERTY sNetId : STRING
GET
sNetId := _sNetId;
END_GET
SET
_sNetId := sNetId;
END_SET
END_PROPERTY

PROPERTY sPath : STRING
GET
sPath := _sPath;
END_GET
SET
_sPath := sPath;
END_SET
END_PROPERTY

METHOD PUBLIC Write : BOOL
VAR_INPUT
	sFileName	: T_MaxString;
	pData 		: PVOID;
	nLength 	: UDINT;
END_VAR
Write := FALSE;
CASE eWriteState OF
	E_FileIoState.READY:
		fbFileOpen(sNetId := _sNetId, bExecute := FALSE);
		fbFileWrite(sNetId := _sNetId, bExecute := FALSE);
		fbFileClose(sNetId := _sNetId, bExecute := FALSE);
		fbCreateDir(sNetId := _sNetId, bExecute := FALSE);
		eWriteState := E_FileIoState.OPEN;
		
	E_FileIoState.OPEN:
		nErrorId := 0;
		IF nHFile = 0 THEN
			fbFileOpen.sPathName := sFileName;
			fbFileOpen.nMode := FOPEN_MODEWRITE;
			fbFileOpen.ePath := PATH_GENERIC;
			fbFileOpen(bExecute := TRUE);
		END_IF
		IF fbFileOpen.hFile <> 0 AND NOT fbFileOpen.bBusy AND NOT fbFileOpen.bError THEN
			nHFile := fbFileOpen.hFile;
			fbFileOpen(bExecute := FALSE);					
			fbFileWrite.hFile := nHFile;
			fbFileWrite.cbWriteLen := nLength;
			fbFileWrite.pWriteBuff := pData;
			eWriteState := E_FileIoState.WRITE;
		END_IF
		IF fbFileOpen.bError THEN
			fbFileOpen(bExecute := FALSE);
			nErrorId := fbFileOpen.nErrId;
			eWriteState := E_FileIoState.CREATE;			
		END_IF
		
	E_FileIoState.CREATE:
		fbCreateDir.sPathName:= _sPath;
		fbCreateDir.ePath:= PATH_GENERIC;
		fbCreateDir(bExecute := TRUE);
		IF NOT fbCreateDir.bBusy AND NOT fbCreateDir.bError THEN
			nErrorId := 0;
			fbCreateDir(bExecute := FALSE);
			eWriteState := E_FileIoState.OPEN;
		END_IF
		IF fbCreateDir.bError THEN
			nErrorId := fbCreateDir.nErrId;
			eWriteState := E_FileIoState.ERROR;			
		END_IF
				
	E_FileIoState.WRITE:
		fbFileWrite(bExecute := TRUE);
		IF NOT fbFileWrite.bBusy AND fbFileWrite.cbWrite = nLength AND NOT fbFileWrite.bError THEN
			fbFileWrite(bExecute := FALSE);
			eWriteState := E_FileIoState.CLOSE;
		END_IF
		IF fbFileWrite.bError THEN
			nErrorId := fbFileWrite.nErrId;
			eWriteState := E_FileIoState.ERROR;
		END_IF
		
	E_FileIoState.CLOSE:
		IF  nHFile <> 0 THEN
			fbFileClose(hFile := nHFile, bExecute := TRUE);
		END_IF
		IF NOT fbFileClose.bBusy THEN
			fbFileClose(bExecute := FALSE);
			nHFile := 0;
			eWriteState := E_FileIoState.READY;
			Write := TRUE;
		END_IF

	E_FileIoState.ERROR:
		F_LogError(CONCAT('Error reading/writing file in ', CONCAT(_sNetId, CONCAT(' - ', _sPath))));
		eWriteState := E_FileIoState.CLOSE;	

END_CASE
END_METHOD

END_FUNCTION_BLOCK

// Common/System/F_LogError
{attribute 'hide_all_locals'}
FUNCTION F_LogError : BOOL
VAR_INPUT
	sMessage : T_MAXSTRING;
END_VAR

VAR CONSTANT	
	LOGHEADER		: T_MAXSTRING := 'Open Commissioning: %s';
END_VAR

ADSLOGSTR(ADSLOG_MSGTYPE_ERROR, LOGHEADER, sMessage);

END_FUNCTION

// Common/Links/FB_LinkDataByte
FUNCTION_BLOCK FB_LinkDataByte EXTENDS FB_LinkDevice
VAR	
	{attribute 'simulation_interface'}
	ControlData		AT %Q* : BYTE;
	{attribute 'simulation_interface'}
	StatusData		AT %I* : BYTE;
END_VAR

SUPER^();

METHOD INTERNAL GetLinkControlData : BYTE
GetLinkControlData := ControlData;
END_METHOD

METHOD INTERNAL SetLinkStatusData : BOOL
VAR_INPUT
	nStatusData : BYTE;
END_VAR
StatusData := nStatusData;
END_METHOD

END_FUNCTION_BLOCK

// Common/Links/FB_LinkDevice
FUNCTION_BLOCK FB_LinkDevice EXTENDS FB_Base
VAR		
	{attribute 'simulation_interface'}
	Status		AT %I* : BYTE;
	{attribute 'simulation_interface'}
	Control		AT %Q* : BYTE;
END_VAR

SUPER^();

METHOD INTERNAL GetControl : BYTE
GetControl := Control;
END_METHOD

METHOD INTERNAL SetStatus : BOOL
VAR_INPUT
	nStatus : BYTE;
END_VAR
Status := nStatus;
END_METHOD

END_FUNCTION_BLOCK

// Common/System/FB_Base
FUNCTION_BLOCK FB_Base

F_IsSystemValid();

END_FUNCTION_BLOCK

// Common/System/F_IsSystemValid
FUNCTION F_IsSystemValid : BOOL
VAR_STAT
	{attribute 'hide'}
	fbTcConfig		: TC_Config;	
	{attribute 'hide'}
	bIsRequested 	: BOOL;
	{attribute 'hide'}
	bIsSystemValid	: BOOL;
END_VAR

IF NOT bIsRequested THEN
	IF NOT __ISVALIDREF(GVL_Core.refSystem) THEN	
		ADSLOGSTR(msgCtrlMask := ADSLOG_MSGTYPE_ERROR OR ADSLOG_MSGTYPE_MSGBOX, 'OC: %s', 'FB_System can not be found! TwinCAT is switched to Config Mode');
		fbTcConfig(NETID := '', SET := TRUE);
		bIsSystemValid := FALSE;
	ELSE
		bIsSystemValid := TRUE;
	END_IF
END_IF

bIsRequested := TRUE;
F_IsSystemValid := bIsSystemValid;

END_FUNCTION

// Common/System/FB_System
{attribute 'reflection'} 
FUNCTION_BLOCK FB_System
VAR_INPUT
	fbAdsMessageHandler 	: FB_AdsMessageHandler;
	fbRecordData 			: FB_RecordData(refAdsMessageHandler := fbAdsMessageHandler);
END_VAR

VAR
	{attribute 'simulation_interface'}
	Control				AT %Q* : BYTE;
	{attribute 'simulation_interface'}
	Status				AT %I* : BYTE;
	{attribute 'simulation_interface'}
	TimeScaling			AT %I* : REAL := 1.0;
	
	{attribute 'instance-path'} 
    {attribute 'noinit'} 
	_sPath 				: STRING;
	
	_bDebug				: BOOL;
	_bVerbose			: BOOL;
	_fDeltaTime 		: REAL;
	_fTimeScaling 		: REAL;
	_eControllerType	: E_ControllerType;
	
	fbPing				: FB_Ping;
	
	{attribute 'hide'}
	fbGetCurTaskIdx 	: TC2_SYSTEM.GETCURTASKINDEX;
END_VAR

InitRun();
fTimeScaling := TimeScaling;
fbPing(bFeedback := Status.7, bTrigger => Control.7);

fbRecordData(); //Execution order -1 relative to FB_AdsMessageHandler
fbAdsMessageHandler();

PROPERTY bDebug : BOOL
GET
bDebug := _bDebug;
END_GET
SET
_bDebug := bDebug;
END_SET
END_PROPERTY

PROPERTY bVerbose : BOOL
GET
bVerbose := _bVerbose;
END_GET
SET
_bVerbose := bVerbose;
END_SET
END_PROPERTY

PROPERTY eControllerType : E_ControllerType
GET
eControllerType := _eControllerType;
END_GET
SET
_eControllerType := eControllerType;
END_SET
END_PROPERTY

PROPERTY PUBLIC fDeltaTime : REAL
GET
fDeltaTime := _fDeltaTime;
END_GET
SET
PRIVATE
_fDeltaTime := fDeltaTime;
END_SET
END_PROPERTY

PROPERTY PUBLIC fTimeScaling : REAL
GET
fTimeScaling := _fTimeScaling;
END_GET
SET
IF fTimeScaling = 0 THEN
	_fTimeScaling := 1.0;
ELSE
	_fTimeScaling := LIMIT(0.01000001, fTimeScaling, 100.0);	
END_IF
END_SET
END_PROPERTY

METHOD PRIVATE InitRun
VAR_INST
	bInitRun 			: BOOL := TRUE;
	sMessageFormat   	: T_MAXSTRING := '%s %s';
	sMessage  			: T_MAXSTRING;
	fbFormatString 		: FB_FormatString;
END_VAR
IF NOT bInitRun THEN RETURN; END_IF
bInitRun := FALSE;

IF __ISVALIDREF(GVL_Core.refSystem) THEN	
	fbFormatString(sFormat := sMessageFormat, arg1 := F_STRINGEx(_sPath), arg2 := F_STRINGEx('FB_System has no single instance! Check the PROGRAM declaration'), sOut => sMessage);
	ADSLOGSTR(msgCtrlMask := ADSLOG_MSGTYPE_ERROR, '%s', sMessage);	
ELSE 
	GVL_Core.refSystem REF= THIS^;
END_IF

fbGetCurTaskIdx();
_fDeltaTime := UDINT_TO_REAL(TwinCAT_SystemInfoVarList._TaskInfo[fbGetCurTaskIdx.index].CycleTime / 10000) / 1000.0;
_fTimeScaling := 1;

fbRecordData.eControllerType := _eControllerType;
END_METHOD

END_FUNCTION_BLOCK

// Common/RecordData/FB_RecordData
{attribute 'conditionalshow_all_locals}
FUNCTION_BLOCK PUBLIC FB_RecordData IMPLEMENTS I_RecordData
VAR_INPUT
	bDisable 				: BOOL; //Deactivate cyclical execution
	bVerbose 				: BOOL; //Log ADS messages data in the console
	eControllerType 		: E_ControllerType; //The data processing logic depends on the controller type	
END_VAR

VAR	
	refAdsMessageHandler	: REFERENCE TO FB_AdsMessageHandler;	
	nDeviceCount			: INT;
	aDeviceList				: ARRAY[0..255] OF UDINT; //The internal device list is used for assistance services. Do not delete or change. 
END_VAR

IF bDisable THEN RETURN; END_IF

//Send WriteRes if last WriteInd has not been read by any device
IF refAdsMessageHandler.stAdsMessageWrite.tPort <> 0 THEN
	SendWriteResponse(refAdsMessageHandler.stAdsMessageRead);
	refAdsMessageHandler.stAdsMessageWrite.tPort := 0;
END_IF

//Send ReadRes if last ReadInd has not been read by any device
IF refAdsMessageHandler.stAdsMessageRead.tPort <> 0 THEN
	SendReadResponse(refAdsMessageHandler.stAdsMessageRead);
	refAdsMessageHandler.stAdsMessageRead.tPort := 0;
END_IF 

(*Ads Message Comments*)
//tNetId			: T_AmsNetID;
//tPort				: T_AmsPort;
//nInvokeId			: UDINT; //Hil: Byte0 and 1 = Port, Byte2 = Subslot, Byte3 = Slot. Sil: ignored.
//nIndexGroup		: UDINT; //16#80000000 + RecordIndex
//nIndexOffset		: UDINT; //Hil: LowWord = SubSlot, HighWord = Slot. Sil: LowWord = HardwareId, HighWord = PlcId.
//nLengthData		: UDINT;
//nResult			: UDINT;
//aData				: ARRAY[0..239] OF BYTE;

METHOD PRIVATE CmpIGrp : BOOL
VAR_INPUT
	nIGrpDevice 	: UDINT;
	nIGrpReceived 	: UDINT;
END_VAR
(* Compare low word only *)
CmpIGrp := (nIGrpDevice AND 16#0000FFFF) = (nIGrpReceived AND 16#0000FFFF) OR nIGrpDevice = 0;
END_METHOD

METHOD PRIVATE CmpInvokeId : BOOL
VAR_INPUT
	nInvokeIdDevice 	: UDINT;
	nInvokeIdReceived 	: UDINT;
END_VAR
IF eControllerType = E_ControllerType.PlcSimAdvanced THEN
	CmpInvokeId := TRUE;
	RETURN;
END_IF

(* Compare low word only. low word = port *)
CmpInvokeId := (nInvokeIdDevice AND 16#0000FFFF) = (nInvokeIdReceived AND 16#0000FFFF);
END_METHOD

METHOD PRIVATE CmpIOffs : BOOL
VAR_INPUT
	nIOffsDevice 	: UDINT;
	nIOffsReceived 	: UDINT;
END_VAR
CmpIOffs := nIOffsDevice = nIOffsReceived OR nIOffsDevice = 16#FFFFFFFF;
END_METHOD

METHOD INTERNAL DataValid : BOOL
VAR_INPUT
	refDeviceAdsMessage 	: REFERENCE TO ST_AdsMessage;
	refHandlerAdsMessage	: REFERENCE TO ST_AdsMessage;
END_VAR
DataValid := FALSE;

IF refHandlerAdsMessage.tPort = 0 THEN
	RETURN;
END_IF

IF NOT CmpInvokeId(refDeviceAdsMessage.nInvokeId, refHandlerAdsMessage.nInvokeId) THEN
	RETURN;
END_IF

IF NOT CmpIOffs(refDeviceAdsMessage.nIdxOffs, refHandlerAdsMessage.nIdxOffs) THEN
	RETURN;
END_IF

IF NOT CmpIGrp(refDeviceAdsMessage.nIdxGrp, refHandlerAdsMessage.nIdxGrp) THEN
	RETURN;
END_IF

(* Copy the received telegram *)
MEMCPY(ADR(refDeviceAdsMessage), ADR(refHandlerAdsMessage), SIZEOF(ST_AdsMessage));

(* Indicate that the telegram has been read by a device
   -> the device is now responsible for the response! *)
refHandlerAdsMessage.tPort := 0;

DataValid := TRUE;
END_METHOD

METHOD FB_init : BOOL
VAR_INPUT
	bInitRetains 				: BOOL; // if TRUE, the retain variables are initialized (warm start / cold start)
	bInCopyCode 				: BOOL;  // if TRUE, the instance afterwards gets moved into the copy code (online change)
	refAdsMessageHandler		: REFERENCE TO FB_AdsMessageHandler;
END_VAR
THIS^.refAdsMessageHandler REF= refAdsMessageHandler;
END_METHOD

(*Try to get a valid ADR read message. If the message is valid, the data in the input structure will be overwritten*)
METHOD PUBLIC GetReadIndication : BOOL
VAR_INPUT
	refDeviceAdsMessage : REFERENCE TO ST_AdsMessage; //Reference ADS Message
END_VAR
IF NOT refAdsMessageHandler.bIsAdsMessageReadValid THEN
	GetReadIndication := FALSE;
	RETURN; 
END_IF

GetReadIndication := DataValid(refDeviceAdsMessage, refAdsMessageHandler.stAdsMessageRead);
END_METHOD

(*Try to get a valid ADR write message. If the message is valid, the data in the input structure will be overwritten*)
METHOD PUBLIC GetWriteIndication : BOOL
VAR_INPUT
	refDeviceAdsMessage : REFERENCE TO ST_AdsMessage; //Reference ADS Message	
END_VAR
IF NOT refAdsMessageHandler.bIsAdsMessageWriteValid THEN
	GetWriteIndication := FALSE;
	RETURN; 
END_IF

GetWriteIndication := DataValid(refDeviceAdsMessage, refAdsMessageHandler.stAdsMessageWrite);
END_METHOD

(*Send ADS Read Response message*)
METHOD PUBLIC SendReadResponse : HRESULT
VAR_INPUT
	stAdsMessage : ST_AdsMessage; //Response ADS Message
END_VAR
CASE eControllerType OF		
	E_ControllerType.PlcSimAdvanced :
		stAdsMessage.nResult := SHR(stAdsMessage.nIdxOffs, 16) + 16#80000000;
END_CASE

SendReadResponse := refAdsMessageHandler.SendReadResponse(stAdsMessage);
END_METHOD

(*Send ADS Write Response message*)
METHOD PUBLIC SendWriteResponse : HRESULT
VAR_INPUT
	stAdsMessage : ST_AdsMessage; //Response ADS Message
END_VAR
CASE eControllerType OF		
	E_ControllerType.PlcSimAdvanced :
		stAdsMessage.nResult := SHR(stAdsMessage.nIdxOffs, 16) + 16#80000000;
END_CASE

SendWriteResponse := refAdsMessageHandler.SendWriteResponse(stAdsMessage);
END_METHOD

(*Subscribe the RecordIdent device to the RecordData services. The RecordIdent device is initialised during subscription*)
METHOD PUBLIC Subscribe
VAR_INPUT
	pRecordIdent	: POINTER TO ST_RecordIdent; //Pointet to RecordIdent Device
	stAdsMessage 	: REFERENCE TO ST_AdsMessage; //Reference to the initial ADS message configuration of the device
END_VAR
IF nDeviceCount > 255 THEN
	F_LogError('More than 256 RecordData devices');
	RETURN;
END_IF

CASE eControllerType OF
	E_ControllerType.NotDefined :	
		stAdsMessage.nInvokeId := pRecordIdent^.nPort + UINT_TO_USINT(pRecordIdent^.nSubSlot) * 16#10000 + UINT_TO_USINT(pRecordIdent^.nSlot) * 16#1000000;		
		stAdsMessage.nIdxOffs := pRecordIdent^.nSubSlot + pRecordIdent^.nSlot * 16#10000;	
		
		IF stAdsMessage.nInvokeId = 0 THEN
			RETURN;
		END_IF
		
		aDeviceList[nDeviceCount] := stAdsMessage.nInvokeId;
	
	E_ControllerType.PlcSimAdvanced :
		stAdsMessage.nIdxOffs := pRecordIdent^.nHardwareId + pRecordIdent^.nPlcId * 16#10000;
		
		IF stAdsMessage.nIdxOffs = 0 THEN
			RETURN;
		END_IF
		
		aDeviceList[nDeviceCount] := stAdsMessage.nIdxOffs;
END_CASE	

nDeviceCount := nDeviceCount + 1;
END_METHOD

END_FUNCTION_BLOCK

// Common/RecordData/I_RecordData
{attribute 'conditionalshow'}
INTERFACE I_RecordData

(*Try to get a valid ADR read message. If the message is valid, the data in the input structure will be overwritten*)
METHOD GetReadIndication : BOOL
VAR_INPUT
	refDeviceAdsMessage : REFERENCE TO ST_AdsMessage; //Reference ADS Message
END_VAR
END_METHOD

(*Try to get a valid ADR write message. If the message is valid, the data in the input structure will be overwritten*)
METHOD GetWriteIndication : BOOL
VAR_INPUT
	refDeviceAdsMessage : REFERENCE TO ST_AdsMessage; //Reference ADS Message
END_VAR
END_METHOD

(*Send ADS Read Response message*)
METHOD SendReadResponse : HRESULT
VAR_INPUT
	stAdsMessage : ST_AdsMessage; //Response ADS Message
END_VAR
END_METHOD

(*Send ADS Write Response message*)
METHOD SendWriteResponse : HRESULT
VAR_INPUT
	stAdsMessage : ST_AdsMessage; //Response ADS Message
END_VAR
END_METHOD

(*Subscribe the RecordIdent device to the RecordData services. The RecordIdent device is initialised during subscription*)
METHOD Subscribe
VAR_INPUT
	pRecordIdent	: POINTER TO ST_RecordIdent; //Pointet to RecordIdent Device
	stAdsMessage 	: REFERENCE TO ST_AdsMessage; //Reference to the initial ADS message configuration of the device
END_VAR
END_METHOD

END_INTERFACE

// Common/Links/FB_LinkDataDWord
FUNCTION_BLOCK FB_LinkDataDWord EXTENDS FB_LinkDevice
VAR		
	{attribute 'simulation_interface'}
	ControlData		AT %Q* : DWORD;
	{attribute 'simulation_interface'}
	StatusData		AT %I* : DWORD;
END_VAR

SUPER^();

METHOD INTERNAL GetLinkControlData : DWORD
GetLinkControlData := ControlData;
END_METHOD

METHOD INTERNAL SetLinkStatusData : BOOL
VAR_INPUT
	nStatusData : DWORD;
END_VAR
StatusData := nStatusData;
END_METHOD

END_FUNCTION_BLOCK

// Common/Links/FB_LinkDataLWord
FUNCTION_BLOCK FB_LinkDataLWord EXTENDS FB_LinkDevice
VAR	
	{attribute 'simulation_interface'}
	ControlData		AT %Q* : LWORD;
	{attribute 'simulation_interface'}
	StatusData		AT %I* : LWORD;
END_VAR

SUPER^();

METHOD INTERNAL GetLinkControlData : LWORD
GetLinkControlData := ControlData;
END_METHOD

METHOD INTERNAL SetLinkStatusData : BOOL
VAR_INPUT
	nStatusData : LWORD;
END_VAR
StatusData := nStatusData;
END_METHOD

END_FUNCTION_BLOCK

// Common/Links/FB_LinkDataReal
FUNCTION_BLOCK FB_LinkDataReal EXTENDS FB_LinkDevice
VAR	
	{attribute 'simulation_interface'}
	ControlData			AT %Q* : REAL;
	{attribute 'simulation_interface'}
	StatusData			AT %I* : REAL;
END_VAR

SUPER^();

METHOD INTERNAL GetLinkControlData : REAL
GetLinkControlData := ControlData;
END_METHOD

METHOD INTERNAL SetLinkStatusData : BOOL
VAR_INPUT
	fStatusData : REAL;
END_VAR
StatusData := fStatusData;
END_METHOD

END_FUNCTION_BLOCK

// Common/Links/FB_LinkDataWord
FUNCTION_BLOCK FB_LinkDataWord EXTENDS FB_LinkDevice
VAR	
	{attribute 'simulation_interface'}
	StatusData		AT %I* : WORD;
	{attribute 'simulation_interface'}
	ControlData		AT %Q* : WORD;
END_VAR

SUPER^();

METHOD INTERNAL GetLinkControlData : WORD
GetLinkControlData := ControlData;
END_METHOD

METHOD INTERNAL SetLinkStatusData : BOOL
VAR_INPUT
	nStatusData : WORD;
END_VAR
StatusData := nStatusData;
END_METHOD

END_FUNCTION_BLOCK

// Common/Utils/F_Clamp01
FUNCTION F_Clamp01 : REAL
VAR_INPUT
	fValue : REAL;
END_VAR

F_Clamp01:= LIMIT(0, fValue, 1);

END_FUNCTION

// Common/Utils/F_GetHByte
FUNCTION F_GetHByte : BYTE
VAR_INPUT
	nWord	: WORD;
END_VAR

F_GetHByte := WORD_TO_BYTE(SHR(nWord, 8));

END_FUNCTION

// Common/Utils/F_GetLByte
FUNCTION F_GetLByte : BYTE
VAR_INPUT
	nWord	: WORD;
END_VAR

F_GetLByte := WORD_TO_BYTE(nWord);

END_FUNCTION

// Common/Utils/F_InverBytesOrder
FUNCTION F_InverBytesOrder : BOOL
VAR_INPUT
	data 	: ANY;
END_VAR

VAR	
	i 		: UDINT;
	nSize	: UDINT;
	aData 	: ARRAY [0..7] OF BYTE;
END_VAR

nSize := DINT_TO_UDINT(data.diSize);
memcpy(ADR(aData), data.pValue, nSize);

FOR i:= 1 TO nSize DO	
	memcpy(data.pValue + i - 1, ADR(aData) + nSize - i, 1);
END_FOR

END_FUNCTION

// Common/Utils/F_Norm
FUNCTION F_Norm : REAL
VAR_INPUT
	fMin 		: REAL;
	fMax 		: REAL;
	fValue 		: REAL;
END_VAR

F_Norm := F_Clamp01((fValue - fMin)/(fMax - fMin));

END_FUNCTION

// Common/Utils/F_ScaleLREAL
FUNCTION F_ScaleLREAL : LREAL
VAR_INPUT
	fValue 		: LREAL;
	fInputMin 	: LREAL;
	fInputMax 	: LREAL;
	fOutputMin 	: LREAL;
	fOutputMax 	: LREAL;
END_VAR

VAR
	fNormalized : LREAL;
END_VAR

VAR_OUTPUT
	bError 		: BOOL;
END_VAR

bError := (fInputMin >= fInputMax) OR (fOutputMin >= fOutputMax);

IF bError THEN
	F_ScaleLREAL := 0.0;
	RETURN;
END_IF

IF fValue < fInputMin THEN
	fNormalized := 0.0;
ELSIF fValue > fInputMax THEN
	fNormalized := 1.0;
ELSE
	fNormalized := (fValue - fInputMin) / (fInputMax - fInputMin);
END_IF

F_ScaleLREAL := fNormalized * (fOutputMax - fOutputMin) + fOutputMin;

END_FUNCTION

// Devices/Basic/FB_Button
FUNCTION_BLOCK FB_Button EXTENDS FB_LinkDevice 
VAR_INPUT
	bEnable		: BOOL; //0-Lamp OFF, 1-Lamp ON
END_VAR

VAR_OUTPUT
	bValue		: BOOL; //0-Released, 1-Pressed
END_VAR

SUPER^();
Control.0 := bEnable;
bValue := Status.0;

END_FUNCTION_BLOCK

// Devices/Basic/FB_Cylinder
FUNCTION_BLOCK FB_Cylinder EXTENDS FB_LinkDevice 
VAR_INPUT
	bRetract : BOOL; //Move to MIN
	bExtend : BOOL; //Move to MAX
END_VAR

VAR_OUTPUT
	bRetracted : BOOL; //Is in MIN
	bExtended : BOOL; //Is in MAX
END_VAR

SUPER^();
bRetracted := Status.0;
bExtended := Status.1;
Control.0 := bRetract;
Control.1 := bExtend;

END_FUNCTION_BLOCK

// Devices/Basic/FB_Device
FUNCTION_BLOCK FB_Device EXTENDS FB_LinkDevice
VAR_INPUT		
	nControl  			: BYTE;
END_VAR

VAR_OUTPUT
	nStatus  			: BYTE;
END_VAR

SUPER^();
Control := nControl;
nStatus := Status;

END_FUNCTION_BLOCK

// Devices/Basic/FB_DeviceByte
FUNCTION_BLOCK FB_DeviceByte EXTENDS FB_LinkDataByte
VAR_INPUT		
	nControl  			: BYTE;
	nControlData  		: BYTE;
END_VAR

VAR_OUTPUT
	nStatus  			: BYTE;
	nStatusData  		: BYTE;
END_VAR

SUPER^();
Control := nControl;
ControlData := nControlData;
nStatus := Status;
nStatusData := StatusData;

END_FUNCTION_BLOCK

// Devices/Basic/FB_DeviceDWord
FUNCTION_BLOCK FB_DeviceDWord EXTENDS FB_LinkDataDWord
VAR_INPUT		
	nControl  			: BYTE;
	nControlData 		: DWORD;
END_VAR

VAR_OUTPUT
	nStatus  			: BYTE;
	nStatusData  		: DWORD;
END_VAR

SUPER^();
Control := nControl;
ControlData := nControlData;
nStatus := Status;
nStatusData := StatusData;

END_FUNCTION_BLOCK

// Devices/Basic/FB_DeviceLWord
FUNCTION_BLOCK FB_DeviceLWord EXTENDS FB_LinkDataLWord
VAR_INPUT		
	nControl  			: BYTE;
	nControlData  		: LWORD;
END_VAR

VAR_OUTPUT
	nStatus  			: BYTE;
	nStatusData  		: LWORD;
END_VAR

SUPER^();
Control := nControl;
ControlData := nControlData;
nStatus := Status;
nStatusData := StatusData;

END_FUNCTION_BLOCK

// Devices/Basic/FB_DeviceReal
FUNCTION_BLOCK FB_DeviceReal EXTENDS FB_LinkDataReal
VAR_INPUT		
	nControl  			: BYTE;
	fControlData  		: REAL;
END_VAR

VAR_OUTPUT
	nStatus  			: BYTE;
	fStatusData  		: REAL;
END_VAR

SUPER^();
Control := nControl;
ControlData := fControlData;
nStatus := Status;
fStatusData := StatusData;

END_FUNCTION_BLOCK

// Devices/Basic/FB_DeviceWord
FUNCTION_BLOCK FB_DeviceWord EXTENDS FB_LinkDataWord
VAR_INPUT		
	nControl  			: BYTE;
	nControlData  		: WORD;
END_VAR

VAR_OUTPUT
	nStatus  			: BYTE;
	nStatusData  		: WORD;
END_VAR

SUPER^();
Control := nControl;
ControlData := nControlData;
nStatus := Status;
nStatusData := StatusData;

END_FUNCTION_BLOCK

// Devices/Basic/FB_Drive
FUNCTION_BLOCK FB_Drive EXTENDS FB_LinkDataREAL
VAR_INPUT
	nControl  		: BYTE;
	fTargetValue 	: REAL; //Target value to drive
END_VAR

VAR_OUTPUT
	nStatus  		: BYTE;
	fActualValue 	: REAL; //Actual value from drive
END_VAR

SUPER^();
Control := nControl;
ControlData := fTargetValue;
nStatus := Status;
fActualValue := StatusData;

END_FUNCTION_BLOCK

// Devices/Basic/FB_Lamp
FUNCTION_BLOCK FB_Lamp EXTENDS FB_LinkDevice 
VAR_INPUT
	bEnable		: BOOL; //0-Lamp OFF, 1 - Lamp ON
END_VAR

SUPER^();
Control.0 := bEnable;

END_FUNCTION_BLOCK

// Devices/Basic/FB_Lock
FUNCTION_BLOCK FB_Lock EXTENDS FB_LinkDataByte 
VAR_INPUT
	bLock			: BOOL;
	nControlData	: BYTE;
END_VAR

VAR_OUTPUT	
	bClosed 		: BOOL;
	bLocked 		: BOOL; 
	nStatusData		: BYTE;
END_VAR

SUPER^();
Control.0 := bLock;
ControlData := nControlData;

bClosed := Status.0;
bLocked := Status.1;
nStatusData := StatusData;

END_FUNCTION_BLOCK

// Devices/Basic/FB_Panel
FUNCTION_BLOCK FB_Panel EXTENDS FB_LinkDataDWord
VAR_INPUT
	nControlData  			: DWORD;
END_VAR

VAR_OUTPUT	
	nStatusData  			: DWORD;
END_VAR

SUPER^();
ControlData := nControlData;
nStatusData := StatusData;

END_FUNCTION_BLOCK

// Devices/Basic/FB_Reader
FUNCTION_BLOCK FB_Reader EXTENDS FB_LinkDataLWORD
VAR_INPUT
	nControl  		: BYTE;
	nCommand 		: ULINT; //Command ID
END_VAR

VAR_INPUT
	nStatus  		: BYTE;
	nResult			: ULINT; //Result Data
END_VAR

SUPER^();
Control := nControl;
ControlData := ULINT_TO_LWORD(nCommand);
nStatus := Status;
nResult := LWORD_TO_ULINT(StatusData);

END_FUNCTION_BLOCK

// Devices/Basic/FB_Robot
FUNCTION_BLOCK FB_Robot EXTENDS FB_LinkDevice
VAR_INPUT
	nControl  			: BYTE;	
	aJointTarget 		: ARRAY[0..11] OF REAL;	
END_VAR

VAR_OUTPUT
	nStatus  			: BYTE;
	aJointStatus 		: ARRAY[0..11] OF REAL;
END_VAR

VAR
	JointStatus AT %I* 	: ARRAY[0..11] OF REAL; //{simulation-interface}
	JointTarget AT %Q* 	: ARRAY[0..11] OF REAL; //{simulation-interface}
	
	{attribute 'hide'}
	adrData				: LWORD;
	{attribute 'hide'}
	nDataLength 		: UDINT;	
END_VAR

SUPER^();

IF (adrData <> 0) THEN	
	MEMCPY(ADR(aJointTarget), adrData, nDataLength);
END_IF

Control := nControl;
MEMCPY(ADR(JointTarget), ADR(aJointTarget), 12 * 4);
MEMCPY(ADR(aJointStatus), ADR(JointStatus), 12 * 4);
nStatus := Status;

METHOD ConnectJoints : BOOL
VAR_INPUT
	Joints : ANY;
	nJointCount : UDINT;
END_VAR
adrData := Joints.pValue;
nDataLength := LIMIT(0, nJointCount * 4, 12 * 4);
END_METHOD

METHOD INTERNAL GetJointsTarget : ARRAY[0..11] OF REAL;
GetJointsTarget := JointTarget;
END_METHOD

METHOD INTERNAL SetJointsStatus : BOOL
VAR_INPUT
	aJointsStatus : ARRAY[0..11] OF REAL;
END_VAR
JointStatus := aJointsStatus;
END_METHOD

END_FUNCTION_BLOCK

// Devices/Basic/FB_SensorAnalog
FUNCTION_BLOCK FB_SensorAnalog EXTENDS FB_LinkDataReal 
VAR_INPUT
	nControl  		: BYTE;
	stConfig		: ST_ScaleConfig;
END_VAR

VAR_OUTPUT	
	nStatus  		: BYTE;
	nValue			: UINT;
	fValue			: REAL;
END_VAR

SUPER^();
Control := nControl;
fValue := StatusData;
nValue := LREAL_TO_UINT(F_ScaleLREAL(fValue, stConfig.fInputMin, stConfig.fInputMax, stConfig.fOutputMin, stConfig.fOutputMax));
nStatus := Status;

END_FUNCTION_BLOCK

// Devices/Basic/FB_SensorBinary
FUNCTION_BLOCK FB_SensorBinary EXTENDS FB_LinkDevice 
VAR_OUTPUT
	bValue		: BOOL; 
END_VAR

SUPER^();
bValue := Status.0;

END_FUNCTION_BLOCK

// Devices/Basic/FB_Switch
FUNCTION_BLOCK FB_Switch EXTENDS FB_LinkDevice
VAR_INPUT		
	nControl  			: BYTE;
END_VAR

VAR_OUTPUT
	nStatus  			: BYTE;
END_VAR

SUPER^();
Control := nControl;
nStatus := Status;

END_FUNCTION_BLOCK

// Devices/Drives/Encoder/FB_Encoder
FUNCTION_BLOCK FB_Encoder
VAR_INPUT
	fInput 			: REAL; //Input Value [unit] or [unit/s]	
	stConfig 		: ST_EncoderConfig;	
END_VAR

VAR_OUTPUT
	nPosition 		: DINT; //Position [INC]
	fPosition 		: LREAL;
END_VAR

VAR
	fFactorNumDen 	: REAL;
	fFactorDenNum 	: REAL;		
	fValue 			: LREAL;
END_VAR

InitRun();
ControlLogic();

METHOD PRIVATE ControlLogic
IF stConfig.bIsIntegral THEN
	fValue := fValue + (fInput * stConfig.fInputFactor * GVL_Core.fbSystem.fDeltaTime);
ELSE
	fValue := fInput * stConfig.fInputFactor;
END_IF

IF stConfig.fModulo > 0.0 THEN
	fPosition := LREAL_TO_REAL(LMOD(fValue, stConfig.fModulo));
ELSE
	fPosition := fValue;
END_IF

IF stConfig.bInvertIncrementValue THEN
	nPosition := LREAL_TO_DINT(fPosition * -fFactorDenNum);
ELSE		
	nPosition := LREAL_TO_DINT(fPosition * fFactorDenNum);
END_IF
END_METHOD

METHOD PRIVATE InitRun
VAR_INST
	bInitRun : BOOL := TRUE;
END_VAR
IF NOT bInitRun THEN RETURN; END_IF
bInitRun := FALSE;

fFactorNumDen := stConfig.fNumerator / stConfig.fDenominator; // Scaling factor INC to Units ??
fFactorDenNum := stConfig.fDenominator / stConfig.fNumerator; // Scaling factor Units to INC
END_METHOD

END_FUNCTION_BLOCK

// Devices/Drives/FB_DS402/FB_DS402
{attribute 'reflection'} 
FUNCTION_BLOCK FB_DS402 EXTENDS FB_LinkDataREAL 
VAR_INPUT
	bSTO 				: BOOL := TRUE;	
	stControlData 		: ST_DS402_6040h_ControlWord;
	nTargetValue		: DINT;	//[INC]
	{attribute 'unity-ui'}
	stConfig			: ST_DS402Config;	
END_VAR

VAR_OUTPUT
	stStatusData 		: ST_DS402_6041h_StatusWord;
	nPosition			: DINT; //[INC]	
	fPosition 			: REAL; //[unit]
	fVelocity 			: REAL; //[unit/s]
END_VAR

VAR		
	{attribute 'instance-path'} 
    {attribute 'noinit'} 
    sPath 				: STRING; 	
	
	fbStateMachine 		: FB_DS402FSM;	
	
	nControlLink		: BYTE; //Control BYTE to data link
	fTargetValue 		: REAL; //Target value to data link
	nStatusLink			: BYTE; //Status BYTE from data link
	fActualValue 		: REAL; //Actual value from data link	
	
	fEncoderNumDen 		: REAL;
	fEncoderDenNum 		: REAL;	
	fPositionLocal 		: REAL; //[unit]
	fVelocityLocal 		: REAL; //[unit/s]	
	
	pControlData		: POINTER TO BYTE; //Addr. Process Output (PO), 6 BYTES FROM FIELDBUS
	pStatusData			: POINTER TO BYTE; //Addr. Process Input (PI), 6 BYTES FROM FIELDBUS
END_VAR

SUPER^();
InitRun();

GetControlData(stControlData, pControlData, stConfig.bSwapProcessData);
ControlLogic();
SetStatusData(stStatusData, pStatusData, stConfig.bSwapProcessData);

METHOD PUBLIC AssignAddress
VAR_INPUT
	ControlWord : ANY; //ControlWord from PLC [6 bytes]
	StatusWord : ANY; //StatusWord to PLC [6 bytes]
END_VAR
pControlData := ControlWord.pValue;
pStatusData := StatusWord.pValue;
END_METHOD

METHOD PRIVATE ControlLogic
VAR
	fTargetVelocitySign : REAL;
	fTargetVelocityFactor : REAL;
	fTargetVelocity : REAL;	
END_VAR
nStatusLink := Status;
fActualValue := StatusData;

IF NOT bSTO THEN RETURN; END_IF

fbStateMachine.stControl := stControlData;
fbStateMachine();
stStatusData := fbStateMachine.stStatus;

IF (fbStateMachine._eState = E_DS402State.S4_OperationEnabled) THEN
	CASE stConfig.eControlMode OF
		E_ControlMode.Position: PositionMode();
		E_ControlMode.Speed: SpeedMode();	
	END_CASE
	
	fPosition := fPositionLocal * stConfig.fGearFactor + stConfig.fPositionOffset;
	fVelocity := fVelocityLocal * stConfig.fGearFactor; 
	
	IF stConfig.fEncoderModulo > 0.0 THEN
		fPosition := LREAL_TO_REAL(LMOD(fPosition, stConfig.fEncoderModulo));
	END_IF

	nPosition := REAL_TO_DINT(fPosition * fEncoderDenNum * stConfig.fEncoderOutputFactor);	
	
	CASE stConfig.eLinkControlMode OF
		E_ControlMode.Position: fTargetValue := fPosition * stConfig.fLinkOutputFactor;
		E_ControlMode.Speed: fTargetValue := fVelocity * stConfig.fLinkOutputFactor;	
	END_CASE
END_IF

Control := nControlLink;
ControlData := fTargetValue;
END_METHOD

PROPERTY eState : E_DS402State
GET
eState := fbStateMachine.eState;
END_GET
END_PROPERTY

METHOD PRIVATE GetControlData
VAR_INPUT
	stControl 		: REFERENCE TO ST_DS402_6040h_ControlWord;
	pAddr			: ULINT; //PO adress
	bSwap 			: BOOL; //Swap BE_TO_HOST
END_VAR

VAR
	nControlWord 	: WORD;
	nValue 			: DWORD;
END_VAR
IF pControlData = 0 THEN RETURN; END_IF

MEMCPY(ADR(stControl), pAddr, 2);

IF stConfig.bSwapProcessData THEN
	MEMCPY(ADR(nControlWord), pAddr, 2);
	nControlWord := BE16_TO_HOST(nControlWord);
	MEMCPY(ADR(stControl), ADR(nControlWord), 2);	
	MEMCPY(ADR(nTargetValue), pAddr + 2, 4);
	nTargetValue := DWORD_TO_DINT(HOST_TO_BE32(DINT_TO_DWORD(nTargetValue)));
ELSE
	MEMCPY(ADR(stControl), pAddr, 2);
	MEMCPY(ADR(nTargetValue), pAddr + 2, 4);	
END_IF
END_METHOD

METHOD PRIVATE InitRun
VAR_INST
	bInitRun : BOOL := TRUE;
END_VAR
IF NOT bInitRun THEN RETURN; END_IF
bInitRun := FALSE;

fEncoderNumDen := ABS(stConfig.fEncoderNumerator) / ABS(stConfig.fEncoderDenominator);
fEncoderDenNum := ABS(stConfig.fEncoderDenominator) / ABS(stConfig.fEncoderNumerator);

IF pControlData = 0 OR pStatusData = 0 THEN
	ADSLOGSTR(ADSLOG_MSGTYPE_WARN, '%s', CONCAT(sPath, ' PLC IO is not assigned!'));	
END_IF
END_METHOD

METHOD PRIVATE PositionMode : BOOL
fVelocityLocal := 0;
fPositionLocal := DINT_TO_REAL(nTargetValue) * fEncoderNumDen;
END_METHOD

METHOD PRIVATE SetStatusData
VAR_INPUT
	stStatus 		: ST_DS402_6041h_StatusWord;
	pAddr			: ULINT;
	bSwap 			: BOOL;
END_VAR

VAR
	nStatusWord 	: WORD;
	nValue 			: DINT;
	nTempWord: DWORD;
END_VAR
IF pAddr <= 0 THEN RETURN; END_IF

IF stConfig.bSwapProcessData THEN
	MEMCPY(ADR(nStatusWord), ADR(stStatus), 2);
	nStatusWord := BE16_TO_HOST(nStatusWord);
	MEMCPY(pAddr, ADR(nStatusWord), 2);

	nValue := DWORD_TO_DINT(HOST_TO_BE32(DINT_TO_DWORD(nPosition)));
	MEMCPY(pAddr + 2, ADR(nValue), 4);
ELSE
	MEMCPY(pAddr, ADR(stStatus), 2);
	MEMCPY(pAddr + 2, ADR(nPosition), 4);
END_IF
END_METHOD

METHOD PRIVATE SpeedMode : BOOL
VAR
	fTargetVelocitySign : REAL;
	fTargetVelocityFactor : REAL;
	fTargetVelocity : REAL;	
END_VAR
fTargetVelocity := DINT_TO_REAL(nTargetValue);
fTargetVelocityFactor := F_Norm(0, 80000, ABS(fTargetVelocity));
fVelocityLocal := stConfig.fReferenceVelocity * fTargetVelocityFactor * F_Sign(fTargetVelocity);
fPositionLocal := fPositionLocal +(fVelocityLocal * GVL_Core.fbSystem.fDeltaTime);
END_METHOD

END_FUNCTION_BLOCK

// Devices/Drives/FB_DS402/FB_DS402FSM
FUNCTION_BLOCK FB_DS402FSM
VAR_INPUT
	bModeSpecific 				: BOOL := TRUE;
	bError 						: BOOL;			
	stControl					: ST_DS402_6040h_ControlWord;
END_VAR

VAR_OUTPUT	
	stStatus					: ST_DS402_6041h_StatusWord;	
END_VAR

VAR	
	_eState 					: E_DS402State := E_DS402State.S0_NotReadyToSwitchOn;	
	rTrig_QuickStop 			: R_TRIG;
	rTrig_Reset 				: R_TRIG;
END_VAR

stStatus.b12_OperationModeSpecific := bModeSpecific;

rTrig_QuickStop(CLK := stControl.b2_QuickStop);
rTrig_Reset(CLK := stControl.b7_FaultReset);

CASE _eState OF
	E_DS402State.S0_NotReadyToSwitchOn : S0_NotReadyToSwitchOn();
	E_DS402State.S1_SwitchOnDisabled : S1_SwitchOnDisabled();
	E_DS402State.S2_ReadyToSwitchOn : S2_ReadyToSwitchOn();
	E_DS402State.S3_SwitchedOn : S3_SwitchedOn();
	E_DS402State.S4_OperationEnabled : S4_OperationEnabled();
	E_DS402State.S5_Fault : S5_Fault();	
	E_DS402State.S6_FaultReactionActive : S6_FaultReactionActive();	
	E_DS402State.S7_QuickStopActive : S7_QuickStopActive();			
END_CASE

PROPERTY eState : E_DS402State
GET
eState := _eState;
END_GET
SET
_eState := eState;
END_SET
END_PROPERTY

METHOD PRIVATE IsDisableOperation : BOOL
IsDisableOperation := 
stControl.b0_SwitchOn 
AND stControl.b1_EnableVoltage 
AND stControl.b2_QuickStop 
AND NOT stControl.b3_EnableOperation
AND NOT stControl.b7_FaultReset;
END_METHOD

METHOD PRIVATE IsDisableVoltage : BOOL
IsDisableVoltage := 
NOT stControl.b1_EnableVoltage
AND NOT stControl.b7_FaultReset;
END_METHOD

METHOD PRIVATE IsEnableOperation : BOOL
IsEnableOperation := 
stControl.b0_SwitchOn 
AND stControl.b1_EnableVoltage 
AND stControl.b2_QuickStop 
AND stControl.b3_EnableOperation
AND NOT stControl.b7_FaultReset;
END_METHOD

METHOD PRIVATE IsFaultReset : BOOL
IsFaultReset := rTrig_Reset.Q;
END_METHOD

METHOD PRIVATE IsQuickStop : BOOL
IsQuickStop := 
NOT stControl.b2_QuickStop
AND NOT stControl.b7_FaultReset;
END_METHOD

METHOD PRIVATE IsShutdown : BOOL
IsShutdown := 
NOT stControl.b0_SwitchOn 
AND stControl.b1_EnableVoltage 
AND stControl.b2_QuickStop
AND NOT stControl.b7_FaultReset;
END_METHOD

METHOD PRIVATE IsSwitchOn : BOOL
IsSwitchOn := 
stControl.b0_SwitchOn 
AND stControl.b1_EnableVoltage 
AND stControl.b2_QuickStop
AND NOT stControl.b7_FaultReset;
END_METHOD

PROPERTY nControl : WORD
GET
nControl.0	:= stControl.b0_SwitchOn;					         
nControl.1	:= stControl.b1_EnableVoltage;				      	
nControl.2	:= stControl.b2_QuickStop;					         	
nControl.3	:= stControl.b3_EnableOperation;			     	
nControl.4	:= stControl.b4_OperationModeSpecific;			
nControl.5	:= stControl.b5_OperationModeSpecific;			
nControl.6	:= stControl.b6_OperationModeSpecific;			
nControl.7	:= stControl.b7_FaultReset;					        	
nControl.8	:= stControl.b8_Reserved;					          	
nControl.9	:= stControl.b9_Reserved;					          
nControl.10	:= stControl.b10_Reserved;					         	
nControl.11	:= stControl.b11_Reserved;					         	
nControl.12	:= stControl.b12_Reserved;					         	
nControl.13	:= stControl.b13_Reserved;					         	
nControl.14	:= stControl.b14_Reserved;					         	
nControl.15 := stControl.b15_Reserved;
END_GET
SET
stControl.b0_SwitchOn 					:= 	nControl.0;	
stControl.b1_EnableVoltage				:= 	nControl.1;		
stControl.b2_QuickStop					:= 	nControl.2;		
stControl.b3_EnableOperation			:= 	nControl.3;		
stControl.b4_OperationModeSpecific		:= 	nControl.4;		
stControl.b5_OperationModeSpecific		:= 	nControl.5;		
stControl.b6_OperationModeSpecific		:= 	nControl.6;		
stControl.b7_FaultReset					:= 	nControl.7;		
stControl.b8_Reserved					:= 	nControl.8;		
stControl.b9_Reserved					:= 	nControl.9;		
stControl.b10_Reserved					:= 	nControl.10;		
stControl.b11_Reserved					:= 	nControl.11;		
stControl.b12_Reserved					:= 	nControl.12;		
stControl.b13_Reserved					:= 	nControl.13;		
stControl.b14_Reserved					:= 	nControl.14;		
stControl.b15_Reserved					:= 	nControl.15;
END_SET
END_PROPERTY

PROPERTY nStatus : WORD
GET
nStatus.0 := stStatus.b0_ReadyToSwitchOn; 			
nStatus.1 := stStatus.b1_SwitchedOn; 				
nStatus.2 := stStatus.b2_OperationEnabled;			
nStatus.3 := stStatus.b3_Fault;					
nStatus.4 := stStatus.b4_VoltageEnabled;
nStatus.5 := stStatus.b5_QuickStop;
nStatus.6 := stStatus.b6_SwitchOnDisabled;			
nStatus.7 := stStatus.b7_Warning;					
nStatus.8 := stStatus.b8_Synchranisation;			
nStatus.9 := stStatus.b9_Remote;			
nStatus.10 := stStatus.b10_TargetReached;				
nStatus.11 := stStatus.b11_InternalLimitActive;		
nStatus.12 := stStatus.b12_OperationModeSpecific;			
nStatus.13 := stStatus.b13_OperationModeSpecific;			
nStatus.14 := stStatus.b14_OperationModeSpecific;			
nStatus.15 := stStatus.b15_ClosedLoopActive;
END_GET
END_PROPERTY

METHOD PRIVATE S0_NotReadyToSwitchOn : BOOL
VAR_INPUT
END_VAR
stStatus.b0_ReadyToSwitchOn 		:= FALSE;
stStatus.b1_SwitchedOn 				:= FALSE;
stStatus.b2_OperationEnabled		:= FALSE;
stStatus.b3_Fault					:= FALSE;
stStatus.b4_VoltageEnabled			:= FALSE;
stStatus.b6_SwitchOnDisabled 		:= FALSE;

_eState := E_DS402State.S1_SwitchOnDisabled;
END_METHOD

METHOD PRIVATE S1_SwitchOnDisabled : BOOL
VAR_INPUT
END_VAR
stStatus.b0_ReadyToSwitchOn 		:= FALSE;
stStatus.b1_SwitchedOn				:= FALSE;
stStatus.b2_OperationEnabled 		:= FALSE;
stStatus.b3_Fault 					:= FALSE;
stStatus.b4_VoltageEnabled			:= FALSE;
stStatus.b6_SwitchOnDisabled 		:= TRUE;

IF IsShutdown() THEN
	_eState := E_DS402State.S2_ReadyToSwitchOn;
END_IF
END_METHOD

METHOD PRIVATE S2_ReadyToSwitchOn : BOOL
VAR_INPUT
END_VAR
stStatus.b0_ReadyToSwitchOn 		:= TRUE;
stStatus.b1_SwitchedOn 				:= FALSE;
stStatus.b2_OperationEnabled 		:= FALSE;
stStatus.b3_Fault 					:= FALSE;
stStatus.b4_VoltageEnabled			:= TRUE;
stStatus.b5_QuickStop 				:= TRUE; 
stStatus.b6_SwitchOnDisabled 		:= FALSE;

IF bError THEN
	_eState := E_DS402State.S6_FaultReactionActive;
	RETURN;
END_IF

IF IsDisableVoltage() OR IsQuickStop() THEN
	_eState := E_DS402State.S1_SwitchOnDisabled;
	RETURN;
END_IF

IF IsSwitchOn() THEN
	_eState := E_DS402State.S3_SwitchedOn;
	RETURN;
END_IF
END_METHOD

METHOD PRIVATE S3_SwitchedOn : BOOL
VAR_INPUT
END_VAR
stStatus.b0_ReadyToSwitchOn 		:= TRUE;
stStatus.b1_SwitchedOn 				:= TRUE;
stStatus.b2_OperationEnabled 		:= FALSE;
stStatus.b3_Fault 					:= FALSE;
stStatus.b5_QuickStop 				:= TRUE; 
stStatus.b6_SwitchOnDisabled 		:= FALSE;

IF bError THEN
	_eState := E_DS402State.S6_FaultReactionActive;
	RETURN;
END_IF

IF IsDisableVoltage() OR IsQuickStop() THEN
	_eState := E_DS402State.S1_SwitchOnDisabled;
	RETURN;
END_IF

IF IsShutdown() THEN
	_eState := E_DS402State.S2_ReadyToSwitchOn;
	RETURN;
END_IF

IF IsEnableOperation() THEN
	_eState := E_DS402State.S4_OperationEnabled;
	RETURN;
END_IF
END_METHOD

METHOD PRIVATE S4_OperationEnabled : BOOL
VAR_INPUT
END_VAR
stStatus.b0_ReadyToSwitchOn				:= TRUE;
stStatus.b1_SwitchedOn 					:= TRUE;
stStatus.b2_OperationEnabled 			:= TRUE;
stStatus.b3_Fault 						:= FALSE;
stStatus.b5_QuickStop 					:= TRUE; 
stStatus.b6_SwitchOnDisabled 			:= FALSE;

IF bError THEN
	_eState := E_DS402State.S6_FaultReactionActive;
	RETURN;
END_IF

IF IsDisableVoltage() THEN
	_eState := E_DS402State.S1_SwitchOnDisabled;
	RETURN;
END_IF

IF IsShutdown() THEN
	_eState := E_DS402State.S2_ReadyToSwitchOn;
	RETURN;
END_IF

IF IsQuickStop() THEN
	_eState := E_DS402State.S7_QuickStopActive;
	RETURN;
END_IF

IF IsDisableOperation() THEN
	_eState := E_DS402State.S3_SwitchedOn;
	RETURN;
END_IF
END_METHOD

METHOD PRIVATE S5_Fault : BOOL
VAR_INPUT
END_VAR
stStatus.b0_ReadyToSwitchOn 		:= FALSE;
stStatus.b1_SwitchedOn				:= FALSE;
stStatus.b2_OperationEnabled 		:= FALSE;
stStatus.b3_Fault 					:= TRUE;
stStatus.b6_SwitchOnDisabled 		:= FALSE;

IF IsFaultReset() THEN
	_eState := E_DS402State.S1_SwitchOnDisabled;
	RETURN;
END_IF
END_METHOD

METHOD PRIVATE S6_FaultReactionActive : BOOL
VAR_INPUT
END_VAR
stStatus.b0_ReadyToSwitchOn 		:= TRUE;
stStatus.b1_SwitchedOn 				:= TRUE;
stStatus.b2_OperationEnabled 		:= TRUE;
stStatus.b3_Fault 					:= TRUE;
stStatus.b6_SwitchOnDisabled 		:= FALSE;

_eState := E_DS402State.S5_Fault;
END_METHOD

METHOD PRIVATE S7_QuickStopActive : BOOL
VAR_INPUT
END_VAR
stStatus.b0_ReadyToSwitchOn 		:= TRUE;
stStatus.b1_SwitchedOn 				:= TRUE;
stStatus.b2_OperationEnabled 		:= TRUE;
stStatus.b3_Fault 					:= FALSE;
stStatus.b5_QuickStop 				:= FALSE; 
stStatus.b6_SwitchOnDisabled		:= FALSE;

IF IsDisableVoltage() THEN
	_eState := E_DS402State.S1_SwitchOnDisabled;
	RETURN;
END_IF

IF IsEnableOperation() THEN
	_eState := E_DS402State.S4_OperationEnabled;
	RETURN;
END_IF
END_METHOD

END_FUNCTION_BLOCK

// Devices/Drives/FB_SimMovidrive/FB_SimMovidrivePDO12
{attribute 'reflection'} 
FUNCTION_BLOCK FB_SimMovidrivePDO12 EXTENDS FB_LinkDataReal
VAR_INPUT
	bSTO					: BOOL := TRUE;	
	stControlData			: ST_SimMovidriveControlData;
	stConfig				: ST_SimMovidriveConfig;
END_VAR                 	
                        	
VAR_OUTPUT              	
	stStatusData			: ST_SimMovidriveStatusData;
	fPosition				: REAL;
	fVelocity 				: REAL;
END_VAR

VAR
    {attribute 'instance-path'} 
    {attribute 'noinit'} 
    sPath 					: STRING; 	
	                    	
	fbSimMovitracFSM		: FB_SimMovitracFSM;
	eSimMovidriveMode		: E_SimMovidriveMode := E_SimMovidriveMode.Idle;
	fbDriveControl			: FB_DriveControl;
	                    	
	pControlData			: POINTER TO BYTE; //Addr. Process Output (PO), 12 BYTES FROM FIELDBUS
	pStatusData				: POINTER TO BYTE; //Addr. Process Input (PI), 12 BYTES TO FIELDBUS
END_VAR

SUPER^();
InitRun();

GetControlData(stControlData, pControlData, stConfig.bSwapProcessData);
ControlLogic();
SetStatusData(stStatusData, pStatusData, stConfig.bSwapProcessData);

(*Assign Process Data Objects to device*)
METHOD PUBLIC AssignProcessData : BOOL
VAR_INPUT
	aControlData 		: ANY; //Addr. Process Output (PO), 12 BYTES FROM FIELDBUS
	aStatusData 		: ANY; //Addr. Process Input (PI), 12 BYTES TO FIELDBUS
END_VAR
THIS^.pControlData := aControlData.pValue;
THIS^.pStatusData := aStatusData.pValue;
END_METHOD

METHOD INTERNAL ControlLogic
VAR_INST
	fSetpointVel		: REAL;
	fSetpointAcc		: REAL;
	fSetpointDec		: REAL;
END_VAR
IF SUPER^.Status.7 THEN	
	fbDriveControl.fPosition := SUPER^.StatusData;
END_IF

eSimMovidriveMode := GetControlMode(stControlData);

(* Copy setpoint values *)
	fSetpointVel 	:= stControlData.nVelocity * stConfig.fRatioVelocity; 
	fSetpointAcc 	:= stControlData.nAcceleration * stConfig.fRatioAccDec;
	fSetpointDec 	:= stControlData.nDeceleration * stConfig.fRatioAccDec;

(* Base state of the controller *)
	fbSimMovitracFSM(
		bControllerInhibit:= stControlData.bControllerInhibit, 
		bRapidStop:= stControlData.bRapidStop, 
		bStop:= stControlData.bStop, 
		bHoldControl:= FALSE);

(* Set parameter *)	
	fbDriveControl.fPositionLimitMin := DINT_TO_REAL(stConfig.nSoftwareLimitMin);
	fbDriveControl.fPositionLimitMax := DINT_TO_REAL(stConfig.nSoftwareLimitMax);
	fbDriveControl.fAccMax := stConfig.fDecRapidStop;
	fbDriveControl.fTolerance := 0.1;

(* Evaluate base state *)
	CASE fbSimMovitracFSM.eState OF
		
	(* Coast stop *)
		E_SimMovitracState.ControllerInhibit:
			fbDriveControl.Stop(stConfig.fDecCoastStop);
		
	(* Rapid stop *)
		E_SimMovitracState.RapidStop:
			fbDriveControl.Stop(stConfig.fDecRapidStop);
		
	(* Ramp stop *)
		E_SimMovitracState.Halt:
			fbDriveControl.Stop(stConfig.fDecRampStop);
		
	(* Enable *)
		E_SimMovitracState.Enable:
			CASE eSimMovidriveMode OF
		
			(* Jog mode *)	
				E_SimMovidriveMode.Jog:
					IF stControlData.bJog1 AND NOT stControlData.bJog2 THEN
						fbDriveControl.MoveVelocity(
							fSetpointVel,
							fSetpointAcc,
							fSetpointDec);
					ELSIF NOT stControlData.bJog1 AND stControlData.bJog2 THEN
						fbDriveControl.MoveVelocity(
							-fSetpointVel,
							fSetpointAcc,
							fSetpointDec);
					ELSE
						fbDriveControl.Stop(fSetpointDec);
					END_IF
				
			(* Ref mode *)
				E_SimMovidriveMode.Ref:
					IF stControlData.bStart THEN
						fbDriveControl.MoveAbsolute(0.0,
							fSetpointVel,
							fSetpointAcc,
							fSetpointDec);
					ELSE
						fbDriveControl.Stop(fSetpointDec);
					END_IF
									
			(* Auto mode *)
				E_SimMovidriveMode.Auto:
					IF stControlData.bStart THEN
						fbDriveControl.MoveAbsolute(
							DINT_TO_REAL(stControlData.nTargetPosition),
							fSetpointVel,
							fSetpointAcc,
							fSetpointDec);
					ELSE
						fbDriveControl.Stop(fSetpointDec);
					END_IF	
			END_CASE	
	END_CASE
	
(* Safe Torque Off *)
	IF NOT bSTO THEN
		fbDriveControl.Stop(stConfig.fDecRapidStop);
	END_IF
	
(* Assign values *)
	fPosition := fbDriveControl.fPosition * stConfig.fRatioPosition;
	fVelocity := fbDriveControl.fVelocity;
	THIS^.ControlData := fPosition;
	
(* Status Word *)
	stStatusData.bMotorTurning			:= fbDriveControl.bIsMoving;
	stStatusData.bInverterReady			:= TRUE;
	stStatusData.bReferenced			:= TRUE;
	stStatusData.bTargetPositionReached	:= fbDriveControl.bIsPositionReached;
	stStatusData.bBrakeReleased			:= fbSimMovitracFSM.eState > E_SimMovitracState.ControllerInhibit;
	stStatusData.bError					:= FALSE;
	stStatusData.bLimitSwitchCW			:= REAL_TO_DINT(fbDriveControl.fPosition) >= stConfig.nSoftwareLimitMax;
	stStatusData.bLimitSwitchCCW		:= REAL_TO_DINT(fbDriveControl.fPosition) <= stConfig.nSoftwareLimitMin;
	stStatusData.nStatus				:= 0;

(* Status values *)
	stStatusData.nActPosition			:= REAL_TO_DINT(fbDriveControl.fPosition);
	stStatusData.nActVelocity			:= REAL_TO_UINT(fbDriveControl.fVelocity / stConfig.fRatioVelocity);
	stStatusData.nActCurrent			:= 0;
	stStatusData.nActUnit				:= 0;
END_METHOD

METHOD INTERNAL GetControlData : BOOL
VAR_INPUT
	stControl 		: REFERENCE TO ST_SimMovidriveControlData;
	pAddr			: ULINT; //PO adress
	bSwap 			: BOOL; //Swap BE_TO_HOST
END_VAR

VAR	
	nControlWord 	: WORD;
END_VAR
IF pAddr <= 0 THEN RETURN; END_IF

IF bSwap THEN 
	MEMCPY(ADR(nControlWord), pAddr, 2);
	nControlWord := BE16_TO_HOST(nControlWord);
	MEMCPY(ADR(stControl), ADR(nControlWord), 2);
	
	MEMCPY(ADR(stControl.nTargetPosition), pAddr + 2, 4);
	stControl.nTargetPosition := DWORD_TO_DINT(BE32_TO_HOST(DINT_TO_DWORD(stControl.nTargetPosition)));
	
	MEMCPY(ADR(stControl.nVelocity), pAddr + 6, 2);
	stControl.nVelocity := BE16_TO_HOST(stControl.nVelocity);
	
	MEMCPY(ADR(stControl.nAcceleration), pAddr + 8, 2);
	stControl.nAcceleration := BE16_TO_HOST(stControl.nAcceleration);
	
	MEMCPY(ADR(stControl.nDeceleration), pAddr + 10, 2);
	stControl.nDeceleration := BE16_TO_HOST(stControl.nDeceleration);	
ELSE
	MEMCPY(ADR(stControl), pAddr, 12);
END_IF
END_METHOD

METHOD INTERNAL GetControlMode : E_SimMovidriveMode
VAR_INPUT
	stControl : ST_SimMovidriveControlData;
END_VAR
IF NOT stControl.bModeLow AND NOT stControl.bModeHigh THEN
	GetControlMode := E_SimMovidriveMode.Idle;
ELSIF stControl.bModeLow AND NOT stControl.bModeHigh THEN
	GetControlMode := E_SimMovidriveMode.Jog;
ELSIF NOT stControl.bModeLow AND stControl.bModeHigh THEN
	GetControlMode := E_SimMovidriveMode.Ref;
ELSE
	GetControlMode := E_SimMovidriveMode.Auto;
END_IF
END_METHOD

METHOD INTERNAL InitRun : BOOL
VAR_INST
	bInitRun : BOOL := TRUE;
END_VAR
IF NOT bInitRun THEN RETURN; END_IF
bInitRun := FALSE;

IF pControlData = 0 OR pStatusData = 0 THEN
	ADSLOGSTR(ADSLOG_MSGTYPE_WARN, CONCAT(sPath, ': %s'), 'Plc address not set.');
END_IF
END_METHOD

METHOD INTERNAL SetStatusData
VAR_INPUT
	stStatus 		: ST_SimMovidriveStatusData;
	pAddr			: ULINT;
	bSwap 			: BOOL;
END_VAR

VAR
	nStatusWord 	: WORD;
END_VAR
IF pAddr <= 0 THEN RETURN; END_IF

IF bSwap THEN 
	MEMCPY(ADR(nStatusWord), ADR(stStatus), 2);
	nStatusWord := HOST_TO_BE16(nStatusWord);
	MEMCPY(pAddr, ADR(nStatusWord), 2);
	
	stStatus.nActPosition := DWORD_TO_DINT(HOST_TO_BE32(DINT_TO_DWORD(stStatus.nActPosition)));
	MEMCPY(pAddr + 2, ADR(stStatus.nActPosition), 4);
	
	stStatus.nActVelocity := HOST_TO_BE16(stStatus.nActVelocity);
	MEMCPY(pAddr + 6, ADR(stStatus.nActVelocity), 2);
	
	stStatus.nActCurrent := HOST_TO_BE16(stStatus.nActCurrent);
	MEMCPY(pAddr + 8, ADR(stStatus.nActCurrent), 2);
	
	stStatus.nActUnit := HOST_TO_BE16(stStatus.nActUnit);
	MEMCPY(pAddr + 10, ADR(stStatus.nActUnit), 2);
ELSE
	MEMCPY(pAddr, ADR(stStatus), 12);
END_IF
END_METHOD

END_FUNCTION_BLOCK

// Devices/Drives/FB_SimMovitracFSM/FB_SimMovitracFSM
FUNCTION_BLOCK INTERNAL FB_SimMovitracFSM
VAR_INPUT
	bControllerInhibit	: BOOL;
	bRapidStop			: BOOL;
	bStop				: BOOL;
	bHoldControl		: BOOL;
END_VAR
VAR_OUTPUT
	eState			: E_SimMovitracState := E_SimMovitracState.ControllerInhibit;	
END_VAR

(* Statemachine *)	
	CASE eState OF	
		E_SimMovitracState.ControllerInhibit: ControllerInhibit();		
		E_SimMovitracState.RapidStop:	RapidStop();
		E_SimMovitracState.Halt: Halt();
		E_SimMovitracState.HoldControl: HoldControl();
		E_SimMovitracState.Enable: Enable();
	END_CASE

METHOD INTERNAL ControllerInhibit
VAR_INPUT
END_VAR
(*to RapidStop*)	
	IF NOT bControllerInhibit THEN
		eState := E_SimMovitracState.RapidStop;
	END_IF
END_METHOD

METHOD INTERNAL Enable
VAR_INPUT
END_VAR
(*to ControllerInhibit*)	
	IF bControllerInhibit THEN
		eState := E_SimMovitracState.ControllerInhibit;
		RETURN;
	END_IF

(*to RapidStop*)	
	IF NOT bRapidStop THEN
		eState := E_SimMovitracState.RapidStop;
		RETURN;
	END_IF
	
(*to Halt*)	
	IF NOT bStop THEN
		eState := E_SimMovitracState.Halt;
		RETURN;
	END_IF
	
(*to HoldControl*)	
	IF bHoldControl THEN
		eState := E_SimMovitracState.HoldControl;
	END_IF
END_METHOD

METHOD INTERNAL Halt
VAR_INPUT
END_VAR
(*to ControllerInhibit*)	
	IF bControllerInhibit THEN
		eState := E_SimMovitracState.ControllerInhibit;
		RETURN;
	END_IF

(*to RapidStop*)	
	IF NOT bRapidStop THEN
		eState := E_SimMovitracState.RapidStop;
		RETURN;
	END_IF
	
(*to HoldControl*)	
	IF bStop AND bHoldControl THEN
		eState := E_SimMovitracState.HoldControl;
		RETURN;
	END_IF

(*to Enable*)	
	IF bStop AND NOT bHoldControl THEN
		eState := E_SimMovitracState.Enable;
	END_IF
END_METHOD

METHOD INTERNAL HoldControl
VAR_INPUT
END_VAR
(*to ControllerInhibit*)	
	IF bControllerInhibit THEN
		eState := E_SimMovitracState.ControllerInhibit;
		RETURN;
	END_IF

(*to RapidStop*)	
	IF NOT bRapidStop THEN
		eState := E_SimMovitracState.RapidStop;
		RETURN;
	END_IF
	
(*to Halt*)	
	IF NOT bStop THEN
		eState := E_SimMovitracState.Halt;
		RETURN;
	END_IF
	
(*to Enable*)	
	IF NOT bHoldControl THEN
		eState := E_SimMovitracState.Enable;
	END_IF
END_METHOD

PROPERTY nState : E_SimMovitracState
GET
nState := eState;
END_GET
SET
eState := nState;
END_SET
END_PROPERTY

METHOD INTERNAL RapidStop
VAR_INPUT
END_VAR
(*to ControllerInhibit*)	
	IF bControllerInhibit THEN
		eState := E_SimMovitracState.ControllerInhibit;
		RETURN;
	END_IF

(*to Halt*)	
	IF bRapidStop THEN
		eState := E_SimMovitracState.Halt;
	END_IF
END_METHOD

END_FUNCTION_BLOCK

// Devices/Drives/FB_SimMovitrac/FB_SimMovitrac
{attribute 'reflection'} 
FUNCTION_BLOCK FB_SimMovitrac EXTENDS FB_LinkDataReal
VAR_INPUT
	bSTO					: BOOL := TRUE;
	stControlData			: ST_SimMovitracControlData;
	stConfig				: ST_SimMovitracConfig;	
END_VAR

VAR_OUTPUT
	stStatusData			: ST_SimMovitracStatusData;
	fVelocity 				: REAL;	
END_VAR

VAR
    {attribute 'instance-path'} 
    {attribute 'noinit'} 
    sPath 					: STRING; 
	                		
	fbSimMovitracFSM		: FB_SimMovitracFSM;
	fbDriveControl			: FB_DriveControl;
	                		
	pControlData			: POINTER TO BYTE; //Addr. Process Output (PO), 6 BYTES FROM FIELDBUS
	pStatusData				: POINTER TO BYTE; //Addr. Process Input (PI), 6 BYTES TO FIELDBUS
END_VAR

VAR CONSTANT
	MAX_VALUE_UINT			: UINT := 65535;
END_VAR

SUPER^();
InitRun();

GetControlData(stControlData, pControlData, stConfig.bSwapProcessData);
ControlLogic();
SetStatusData(stStatusData, pStatusData, stConfig.bSwapProcessData);

(*Assign Process Data Objects to device*)
METHOD PUBLIC AssignProcessData : BOOL
VAR_INPUT
	aControlData 		: ANY; //Addr. Process Output (PO), 6 BYTES FROM FIELDBUS
	aStatusData 		: ANY; //Addr. Process Input (PI), 6 BYTES TO FIELDBUS
END_VAR
THIS^.pControlData := aControlData.pValue;
THIS^.pStatusData := aStatusData.pValue;
END_METHOD

METHOD INTERNAL ControlLogic
VAR
	fDecCoastStop	: REAL;
	fDecRapidStop	: REAL;
	fProcessRamp	: REAL;
END_VAR
(* Limit values *)
	stConfig.fDecCoastStop 	:= LIMIT(1, stConfig.fDecCoastStop, MAX_VALUE_UINT);
	stConfig.fDecRapidStop 	:= LIMIT(1, stConfig.fDecRapidStop, MAX_VALUE_UINT);
	stControlData.nSetpointSpeed 	:= LIMIT(-REAL_TO_INT(stConfig.fReferenceVelocity), stControlData.nSetpointSpeed, REAL_TO_INT(stConfig.fReferenceVelocity));
	stControlData.nRamp 			:= LIMIT(1, stControlData.nRamp, MAX_VALUE_UINT);

(* Calculate acceleration / deceleration targets *)
	fDecCoastStop := stConfig.fReferenceVelocity * 1000 / stConfig.fDecCoastStop;
	fDecRapidStop := stConfig.fReferenceVelocity * 1000 / stConfig.fDecRapidStop;
	fProcessRamp := stConfig.fReferenceVelocity * 1000 / UINT_TO_REAL(stControlData.nRamp);
	
(* Base state of the controller *)
	fbSimMovitracFSM(
		bControllerInhibit:= stControlData.bControllerInhibit, 
		bRapidStop:= stControlData.bRapidStop, 
		bStop:= stControlData.bStop, 
		bHoldControl:= FALSE);
	
(* Safe Torque Off *)
IF NOT bSTO THEN
	fbDriveControl.Stop(fDecRapidStop);
ELSE
	
	(* Evaluate base state *)
	CASE fbSimMovitracFSM.eState OF
	(* Coast stop *)
		E_SimMovitracState.ControllerInhibit:
			fbDriveControl.Stop(fDecCoastStop);			
	(* Rapid stop *)
		E_SimMovitracState.RapidStop:
			fbDriveControl.Stop(fDecRapidStop);		
	(* Ramp stop *)
		E_SimMovitracState.Halt:
			fbDriveControl.Stop(fProcessRamp);		
	(* Enable *)		
		E_SimMovitracState.Enable:
			fbDriveControl.MoveVelocity(stControlData.nSetpointSpeed * 0.2, fProcessRamp, fProcessRamp);
	END_CASE
END_IF

(* Velocity value *)
	ControlData := fVelocity := fbDriveControl.fVelocity * stConfig.fGearFactor;
	
(* Status Word *)
	stStatusData.bEnableOutputStage		:= fbDriveControl.fVelocity <> 0;
	stStatusData.bInverterReady   		:= TRUE;
	stStatusData.bPoDataEnable    		:= FALSE;
	stStatusData.bReserved3       		:= FALSE;
	stStatusData.bReserved4       		:= FALSE;
	stStatusData.bError           		:= FALSE;
	stStatusData.bReserved6       		:= FALSE;
	stStatusData.bReserved7       		:= FALSE;
	stStatusData.nStatus				:= 0;

(* Status values *)
	stStatusData.nActSpeed				:= REAL_TO_INT(fbDriveControl.fVelocity / 0.2);
END_METHOD

METHOD INTERNAL GetControlData
VAR_INPUT
	stControl 		: REFERENCE TO ST_SimMovitracControlData;
	pAddr			: ULINT; //PO adress
	bSwap 			: BOOL; //Swap BE_TO_HOST
END_VAR

VAR
	nCtrlIndex		: DWORD;
	nSpeedIndex		: DWORD;
	nRampIndex		: DWORD;
END_VAR
IF pAddr <= 0 THEN RETURN; END_IF

nCtrlIndex := stConfig.nCtrlAssign;
nSpeedIndex := stConfig.nSpeedAssign;
nRampIndex := stConfig.nRampAssign;
	
IF stConfig.bSwapProcessData THEN
	MEMCPY(ADR(stControlData) + 1, pAddr + nCtrlIndex, 1);
	MEMCPY(ADR(stControlData), pAddr + nCtrlIndex + 1, 1);
	MEMCPY(ADR(stControlData.nSetpointSpeed) + 1, pAddr + nSpeedIndex, 1);
	MEMCPY(ADR(stControlData.nSetpointSpeed), pAddr + nSpeedIndex + 1, 1);
	
	IF nRampIndex > E_SimMovitracAssign.ProcessData3 THEN
		MEMCPY(ADR(stControlData.nRamp) + 1, pAddr + nRampIndex, 2);
		MEMCPY(ADR(stControlData.nRamp), pAddr + nRampIndex + 1, 2);
	ELSE
		stControlData.nRamp := REAL_TO_UINT(stConfig.fProcessRamp);
	END_IF
ELSE
	MEMCPY(ADR(stControlData), pControlData + nCtrlIndex, 2);
	MEMCPY(ADR(stControlData.nSetpointSpeed), pAddr + nSpeedIndex, 2);
	
	IF nRampIndex > E_SimMovitracAssign.ProcessData3 THEN
		memcpy(ADR(stControlData.nRamp), pAddr + nRampIndex, 2);
	ELSE
		stControlData.nRamp := REAL_TO_UINT(stConfig.fProcessRamp);
	END_IF			
END_IF
END_METHOD

METHOD INTERNAL InitRun : BOOL
VAR_INST
	bInitRun : BOOL := TRUE;
END_VAR
IF NOT bInitRun THEN RETURN; END_IF
bInitRun := FALSE;

IF pControlData = 0 OR pStatusData = 0 THEN
	ADSLOGSTR(ADSLOG_MSGTYPE_WARN, CONCAT(sPath, ': %s'), 'Plc address not set.');
END_IF

fbDriveControl.fPositionLimitMin := 0;
fbDriveControl.fPositionLimitMax := 0;
fbDriveControl.fAccMax := 0;
fbDriveControl.fTolerance := 0.1;
END_METHOD

METHOD INTERNAL SetStatusData : BOOL
VAR_INPUT
	stStatus 		: ST_SimMovitracStatusData;
	pAddr			: ULINT;
	bSwap 			: BOOL;
END_VAR

VAR
	nStatusIndex	: DWORD;
	nSpeedActIndex	: DWORD;
END_VAR
IF pAddr <= 0 THEN RETURN; END_IF

nStatusIndex := stConfig.nStatusAssign;
nSpeedActIndex := stConfig.nSpeedActAssign;

IF stConfig.bSwapProcessData THEN
	MEMCPY(pAddr + nStatusIndex + 1, ADR(stStatusData), 1);
	MEMCPY(pAddr + nStatusIndex, ADR(stStatusData.nStatus), 1);
	MEMCPY(pAddr + nSpeedActIndex + 1, ADR(stStatusData.nActSpeed), 1);
	MEMCPY(pAddr + nSpeedActIndex, ADR(stStatusData.nActSpeed) + 1, 1);
ELSE	
	MEMCPY(pAddr + nStatusIndex, ADR(stStatusData), 2);
	MEMCPY(pAddr + nSpeedActIndex, ADR(stStatusData.nActSpeed), 2);	
END_IF
END_METHOD

END_FUNCTION_BLOCK

// Devices/Drives/FB_SimMovitrac/FB_SimMovitracB
{attribute 'reflection'} 
FUNCTION_BLOCK FB_SimMovitracB EXTENDS FB_LinkDataReal
VAR_INPUT	
	bSTO 						: BOOL := TRUE;	
	stControlData				: ST_SimMovitracControlData;
	stConfig 					: ST_SimMovitracConfig;	
END_VAR

VAR_OUTPUT
	stStatusData				: ST_SimMovitracStatusData;	 
	fVelocity 					: REAL; //[unit/s]	
END_VAR


VAR
	{attribute 'instance-path'} 
    {attribute 'noinit'} 
    sPath 						: STRING; 	

	fbSimMovitracFSM			: FB_SimMovitracFSM;
	fSetPoint       			: REAL;
	
	pControlData				: POINTER TO BYTE; //Addr. Process Output (PO), 6 BYTES FROM FIELDBUS
	pStatusData					: POINTER TO BYTE; //Addr. Process Input (PI), 6 BYTES TO FIELDBUS
END_VAR

SUPER^();
InitRun();

GetControlData(stControlData, pControlData, stConfig.bSwapProcessData);
ControlLogic();
SetStatusData(stStatusData, pStatusData, stConfig.bSwapProcessData);

(*Assign Process Data Objects to device*)
METHOD PUBLIC AssignProcessData : BOOL
VAR_INPUT
	aControlData 		: ANY; //Addr. Process Output (PO), 6 BYTES FROM FIELDBUS
	aStatusData 		: ANY; //Addr. Process Input (PI), 6 BYTES TO FIELDBUS
END_VAR
THIS^.pControlData := aControlData.pValue;
THIS^.pStatusData := aStatusData.pValue;
END_METHOD

METHOD INTERNAL ControlLogic
fbSimMovitracFSM(bControllerInhibit:= stControlData.bControllerInhibit, bRapidStop:= stControlData.bRapidStop,	bStop:= stControlData.bStop, bHoldControl:= FALSE);

IF bSTO AND fbSimMovitracFSM.eState = E_SimMovitracState.Enable THEN
	fSetPoint := LREAL_TO_REAL(F_ScaleLREAL(INT_TO_REAL(stControlData.nSetpointSpeed), -32767, 32767, -1.0, 1.0));
ELSE
	fSetPoint := 0;
END_IF
	
(* Velocity value *)
	fVelocity := stConfig.fReferenceVelocity * fSetPoint;
	ControlData := fVelocity * stConfig.fGearFactor;
	
